METHOD PROTECTED M_MeasurementClient : BOOL
VAR_INPUT
END_VAR
CASE eFixtureStateMeasure OF
	UNIVERSAL_FIXTURE_MEASURE_SEND_DATA:
		(* Prepare and send data to client *)
		sSendData := CONCAT('START;',UDINT_TO_STRING(iSampleID));
		sSendData := CONCAT(sSendData, '$R$N');
		FUN_StringToTcpBufferData(sMessageAddr := ADR(sSendData), stSendDataAddr := ADR(stSendData));
		fbTcpClient.MR_AppendToSendBuffer(stData := stSendData);
		
		(* Prepare data for logger *)
		IF bUseLogger THEN
			MEMSET(ADR(sLoggerMessage),0,INT_TO_UDINT(LEN(sLoggerMessage)));
			sLoggerMessage := CONCAT('SampleID:',UDINT_TO_STRING(iSampleID));
			
		END_IF
		
		eFixtureStateMeasure := UNIVERSAL_FIXTURE_MEASURE_RECIVE_DATA;
		
	UNIVERSAL_FIXTURE_MEASURE_RECIVE_DATA:
		stReciveData := fbTcpClient.NextRecivedMessage;
		
		IF stReciveData.iLength > 0 THEN
			FUN_TcpBufferDataToString(sMessageAddr := ADR(sRecivedData), stReturnDataAddr := ADR(stReciveData));
			
			(* Sample accepted *)
			IF MEMCMP(ADR(sRecivedData),ADR(sSAMPLE_ACCEPTED),INT_TO_UDINT(LEN(sSAMPLE_ACCEPTED))) = 0 THEN
				IF bUseLogger THEN
					sLoggerMessage := CONCAT(sLoggerMessage,sSAMPLE_ACCEPTED);
					fbMeasurementLogger.MR_AddLogs(sLoggerMessage);
					
				END_IF
				eSampleResult := UNIVERSAL_FIXTURE_SAMPLE_ACCEPTED;
				eFixtureStateMeasure := UNIVERSAL_FIXTURE_MEASURE_DONE;
				
			(* Sample rejected *)
			ELSIF MEMCMP(ADR(sRecivedData),ADR(sSAMPLE_REJECTED),INT_TO_UDINT(LEN(sSAMPLE_REJECTED))) = 0 THEN
				IF bUseLogger THEN
					sLoggerMessage := CONCAT(sLoggerMessage,sSAMPLE_REJECTED);
					fbMeasurementLogger.MR_AddLogs(sLoggerMessage);
					
				END_IF
				eSampleResult := UNIVERSAL_FIXTURE_SAMPLE_REJECTED;
				eFixtureStateMeasure := UNIVERSAL_FIXTURE_MEASURE_DONE;
				
			END_IF
		END_IF
		
	UNIVERSAL_FIXTURE_MEASURE_DONE:
		fbTcpClient.MR_ClearAllBuffers();
		eFixtureStateMeasure := UNIVERSAL_FIXTURE_MEASURE_SEND_DATA;
		eFixtureState := UNIVERSAL_FIXTURE_METHOD_DONE;
		
END_CASE
END_METHOD

METHOD PROTECTED M_MeasurementServer : BOOL
VAR_INPUT
END_VAR
CASE eFixtureStateMeasure OF
	UNIVERSAL_FIXTURE_MEASURE_WAIT_FOR_CLIENT:
		IF fbTcpServer.ServerState = TCPIP_SERVER_RUNNING_DATA_EXCHANGE THEN
			eFixtureStateMeasure := UNIVERSAL_FIXTURE_MEASURE_SEND_DATA;
		END_IF
		
	UNIVERSAL_FIXTURE_MEASURE_SEND_DATA:
		(* Prepare and send data to client *)
		sSendData := CONCAT('START;',UDINT_TO_STRING(iSampleID));
		sSendData := CONCAT(sSendData, '$R$N');
		FUN_StringToTcpBufferData(sMessageAddr := ADR(sSendData), stSendDataAddr := ADR(stSendData));
		fbTcpServer.MR_AppendToSendBuffer(stData := stSendData);
		
		(* Prepare data for logger *)
		IF bUseLogger THEN
			MEMSET(ADR(sLoggerMessage),0,INT_TO_UDINT(LEN(sLoggerMessage)));
			sLoggerMessage := CONCAT('SampleID:',UDINT_TO_STRING(iSampleID));
		END_IF
		
		eFixtureStateMeasure := UNIVERSAL_FIXTURE_MEASURE_RECIVE_DATA;
		
	UNIVERSAL_FIXTURE_MEASURE_RECIVE_DATA:
		stReciveData := fbTcpServer.LastRecivedMessage;
		IF stReciveData.iLength > 0 THEN
			FUN_TcpBufferDataToString(sMessageAddr := ADR(sRecivedData), stReturnDataAddr := ADR(stReciveData));
			
			(* Sample accepted *)
			IF MEMCMP(ADR(sRecivedData),ADR(sSAMPLE_ACCEPTED),INT_TO_UDINT(LEN(sSAMPLE_ACCEPTED))) = 0 THEN
				IF bUseLogger THEN
					sLoggerMessage := CONCAT(sLoggerMessage,sSAMPLE_ACCEPTED);
					fbMeasurementLogger.MR_AddLogs(sLoggerMessage);
				END_IF
				eSampleResult := UNIVERSAL_FIXTURE_SAMPLE_ACCEPTED;
				eFixtureStateMeasure := UNIVERSAL_FIXTURE_MEASURE_DONE;
				
			(* Sample rejected *)
			ELSIF MEMCMP(ADR(sRecivedData),ADR(sSAMPLE_REJECTED),INT_TO_UDINT(LEN(sSAMPLE_REJECTED))) = 0 THEN
				IF bUseLogger THEN
					sLoggerMessage := CONCAT(sLoggerMessage,sSAMPLE_REJECTED);
					fbMeasurementLogger.MR_AddLogs(sLoggerMessage);
				END_IF
				eSampleResult := UNIVERSAL_FIXTURE_SAMPLE_REJECTED;
				eFixtureStateMeasure := UNIVERSAL_FIXTURE_MEASURE_DONE;
				
			END_IF
		END_IF
		
	UNIVERSAL_FIXTURE_MEASURE_DONE:
		fbTcpServer.MR_ClearAllBuffers();
		eFixtureStateMeasure := UNIVERSAL_FIXTURE_MEASURE_WAIT_FOR_CLIENT;
		eFixtureState := UNIVERSAL_FIXTURE_METHOD_DONE;
		
END_CASE
END_METHOD

METHOD MR_Abort : BOOL
IF eFixtureState >= UNIVERSAL_FIXTURE_INITIALIZING THEN
	bBusy := TRUE;
	MR_Abort := FALSE;
	eFixtureState := UNIVERSAL_FIXTURE_ABORTING;
	fbMachineLogger.MR_AddLogs(CONCAT(sName,' : abort requested'));	

ELSIF eFixtureState = UNIVERSAL_FIXTURE_UNINITIALIZED THEN
	bBusy := FALSE;
	MR_Abort := TRUE;
	fbMachineLogger.MR_AddLogs(CONCAT(sName,' : abort done'));	

END_IF
END_METHOD

METHOD MR_Close : BOOL
IF eFixtureState = UNIVERSAL_FIXTURE_IDLE AND THIS^.SocketOpen THEN
	bBusy := TRUE;	
	MR_Close := FALSE;
	eFixtureState := UNIVERSAL_FIXTURE_CLOSE;
	fbMachineLogger.MR_AddLogs(CONCAT(sName,' : close requested'));	
	
ELSIF eFixtureState = UNIVERSAL_FIXTURE_METHOD_DONE THEN
	bBusy := FALSE;
	MR_Close := TRUE;
	fbMachineLogger.MR_AddLogs(CONCAT(sName,' : close done'));	

END_IF
END_METHOD

METHOD MR_FirstCycle : BOOL
VAR_INPUT
	sFixtureName 		: STRING;		(*  *)
	sHost				: T_IPv4Addr;	(*  *)
	sAmsNetID 			: T_AmsNetID;	(*  *)
	iPort				: UINT;			(*  *)
	tTimeout			: TIME;			(*  *)
	bUseLogger			: BOOL;			(*  *)
	bClientConnection 	: BOOL;			(*  *)
	sFileDir			: STRING;		(*  *)
	sFileName			: STRING;		(*  *)
	bCreateFileAtStart	: BOOL;
	bAddHeader			: BOOL;
	bAddTimeStamp		: BOOL;	
END_VAR
THIS^.sName := sFixtureName;
THIS^.bUseLogger := bUseLogger;
THIS^.bClientConnection := bClientConnection;

IF THIS^.bClientConnection THEN 
	(* Set fixture client initial parameters *)
	THIS^.fbTcpClient.MR_FirstCycle(	sName 		:= CONCAT('TCP/IP client of ',sFixtureName),
										sHost		:= sHost,
										sAmsNetID	:= sAmsNetID,
										iPort 		:= iPort,
										tTimeout 	:= tTimeout);	
ELSE
	(* Set fixture server initial parameters *)
	THIS^.fbTcpServer.MR_FirstCycle(	sName 		:= CONCAT('TCP/IP server of ',sFixtureName),
										sHost		:= sHost,
										sAmsNetID	:= sAmsNetID,
										iPort 		:= iPort,
										tTimeout 	:= tTimeout);
END_IF								
									
IF THIS^.bUseLogger THEN
	(* Set measurement logger initial parameters*)									
	THIS^.fbMeasurementLogger.MR_FirstCycle(sName 	:= sName,
											sFileDir 	:= sFileDir,
											sFileName 	:= sFileName,
											sAmsNetId 	:= '',
											bCreateFileAtStart := bCreateFileAtStart,
											bAddHeader 	:= bAddHeader,
											bAddTimeStamp := bAddTimeStamp);	
END_IF
END_METHOD

METHOD MR_Init : BOOL
IF eFixtureState = UNIVERSAL_FIXTURE_UNINITIALIZED THEN
	bBusy := TRUE;
	MR_Init := FALSE;
	
	IF bClientConnection THEN 
		eConnnectionType := UNIVERSAL_FIXTURE_CLIENT_CONNECTION;
		eFixtureStateInit := UNIVERSAL_FIXTURE_INIT_TCP_CLIENT;
		
	ELSE
		eConnnectionType := UNIVERSAL_FIXTURE_SERVER_CONNECTION;	
		eFixtureStateInit := UNIVERSAL_FIXTURE_INIT_TCP_SERVER;	
		
	END_IF
	
	eFixtureState := UNIVERSAL_FIXTURE_INITIALIZING;
	fbMachineLogger.MR_AddLogs(CONCAT(sName,' : initialization requested'));	
	
ELSIF eFixtureState >= UNIVERSAL_FIXTURE_READY THEN
	bBusy := FALSE;
	MR_Init := TRUE;
	fbMachineLogger.MR_AddLogs(CONCAT(sName,' : initialization done'));
	
END_IF
END_METHOD

METHOD MR_Measure : BOOL
VAR_INPUT
	iSampleID : UINT;
END_VAR
IF eFixtureState = UNIVERSAL_FIXTURE_IDLE THEN
	bBusy := TRUE;
	MR_Measure := FALSE;
	THIS^.iSampleID := iSampleID;
	THIS^.eSampleResult := UNIVERSAL_FIXTURE_SAMPLE_UNKNOWN;
	
	IF eConnnectionType = UNIVERSAL_FIXTURE_SERVER_CONNECTION THEN
		eFixtureStateMeasure := UNIVERSAL_FIXTURE_MEASURE_WAIT_FOR_CLIENT;
		
	ELSIF eConnnectionType = UNIVERSAL_FIXTURE_CLIENT_CONNECTION THEN
		eFixtureStateMeasure := UNIVERSAL_FIXTURE_MEASURE_SEND_DATA;
		
	END_IF
	
	eFixtureState := UNIVERSAL_FIXTURE_MEASUREMENT;
	fbMachineLogger.MR_AddLogs(CONCAT(sName,' : measurement requested'));	

ELSIF eFixtureState = UNIVERSAL_FIXTURE_METHOD_DONE THEN
	bBusy := FALSE;
	MR_Measure := TRUE;
	fbMachineLogger.MR_AddLogs(CONCAT(sName,' : measurement done'));	
	
END_IF
END_METHOD

METHOD MR_Open : BOOL
IF eFixtureState = UNIVERSAL_FIXTURE_IDLE AND NOT THIS^.SocketOpen THEN
	bBusy := TRUE;
	MR_Open := FALSE;
	eFixtureState := UNIVERSAL_FIXTURE_OPEN;
	fbMachineLogger.MR_AddLogs(CONCAT(sName,' : open requested'));		
	
ELSIF eFixtureState = UNIVERSAL_FIXTURE_METHOD_DONE THEN
	bBusy := FALSE;
	MR_Open := TRUE;
	fbMachineLogger.MR_AddLogs(CONCAT(sName,' : open done'));		
	
END_IF
END_METHOD

METHOD MR_Reset : BOOL
IF eFixtureState >= UNIVERSAL_FIXTURE_IDLE AND bError THEN
	bBusy := TRUE;
	MR_Reset := FALSE;
	eFixtureState := UNIVERSAL_FIXTURE_RESET;
	fbMachineLogger.MR_AddLogs(CONCAT(sName,' : reset requested'));			
	
ELSIF eFixtureState = UNIVERSAL_FIXTURE_METHOD_DONE THEN
	bBusy := FALSE;
	MR_Reset := TRUE;
	fbMachineLogger.MR_AddLogs(CONCAT(sName,' : reset done'));			
	
END_IF
END_METHOD

METHOD PROTECTED MS_Aborting
VAR_INPUT
END_VAR
CASE eFixtureStateAbort OF
	UNIVERSAL_FIXTURE_ABORT_FILE_LOGGER:
		IF bUseLogger THEN
			fbMeasurementLogger.MR_Abort();
		
			IF NOT fbMeasurementLogger.Busy THEN
				IF eConnnectionType = UNIVERSAL_FIXTURE_SERVER_CONNECTION THEN
					eFixtureStateAbort := UNIVERSAL_FIXTURE_ABORT_TCP_SERVER;
					
				ELSIF eConnnectionType = UNIVERSAL_FIXTURE_CLIENT_CONNECTION THEN
					eFixtureStateAbort := UNIVERSAL_FIXTURE_ABORT_TCP_CLIENT;
					
				END_IF
			END_IF
		ELSE
			IF eConnnectionType = UNIVERSAL_FIXTURE_SERVER_CONNECTION THEN
				eFixtureStateAbort := UNIVERSAL_FIXTURE_ABORT_TCP_SERVER;
				
			ELSIF eConnnectionType = UNIVERSAL_FIXTURE_CLIENT_CONNECTION THEN
				eFixtureStateAbort := UNIVERSAL_FIXTURE_ABORT_TCP_CLIENT;
				
			END_IF
		END_IF
		
	UNIVERSAL_FIXTURE_ABORT_TCP_SERVER:
		fbTcpServer.MR_Abort();
		
		IF NOT fbTcpServer.Active THEN
			eFixtureStateAbort := UNIVERSAL_FIXTURE_ABORT_DONE;
			
		END_IF

	UNIVERSAL_FIXTURE_ABORT_TCP_CLIENT:
		fbTcpClient.MR_Abort();
		
		IF NOT fbTcpClient.Active THEN
			eFixtureStateAbort := UNIVERSAL_FIXTURE_ABORT_DONE;
			
		END_IF
		
	UNIVERSAL_FIXTURE_ABORT_DONE:
		eFixtureStateAbort := UNIVERSAL_FIXTURE_ABORT_FILE_LOGGER;
		eFixtureState := UNIVERSAL_FIXTURE_UNINITIALIZED;
	
END_CASE
END_METHOD

METHOD PROTECTED ABSTRACT MS_Close
VAR_INPUT
END_VAR
;
END_METHOD

METHOD PROTECTED MS_Extension
VAR_INPUT
END_VAR
END_METHOD

METHOD PROTECTED MS_Idle
VAR_INPUT
END_VAR
;
END_METHOD

METHOD PROTECTED MS_Initializing
VAR_INPUT
END_VAR
CASE eFixtureStateInit OF
	UNIVERSAL_FIXTURE_INIT_TCP_SERVER:
		fbTcpServer.MR_Init();
		
		IF fbTcpServer.Active THEN
			eFixtureStateInit := UNIVERSAL_FIXTURE_INIT_FILE_LOGGER;
			
		END_IF

	UNIVERSAL_FIXTURE_INIT_TCP_CLIENT:
		fbTcpClient.MR_Init();
		
		IF fbTcpClient.Active THEN
			eFixtureStateInit := UNIVERSAL_FIXTURE_INIT_FILE_LOGGER;
			
		END_IF
		
	UNIVERSAL_FIXTURE_INIT_FILE_LOGGER:
		IF bUseLogger THEN
			fbMeasurementLogger.MR_Init();
		
			IF fbMeasurementLogger.Busy THEN
				eFixtureStateInit := UNIVERSAL_FIXTURE_INIT_DONE;
				
			END_IF
		ELSE
			eFixtureStateInit := UNIVERSAL_FIXTURE_INIT_DONE;
			
		END_IF
		
	UNIVERSAL_FIXTURE_INIT_DONE:
		eFixtureStateInit := UNIVERSAL_FIXTURE_INIT_TCP_SERVER;
		eFixtureState := UNIVERSAL_FIXTURE_READY;
	
END_CASE
END_METHOD

METHOD PROTECTED MS_Measurement
VAR_INPUT
END_VAR
IF eConnnectionType = UNIVERSAL_FIXTURE_SERVER_CONNECTION THEN
	M_MeasurementServer();
	
ELSIF eConnnectionType = UNIVERSAL_FIXTURE_CLIENT_CONNECTION THEN
	M_MeasurementClient();
	
END_IF
END_METHOD

METHOD PROTECTED MS_MethodDone
VAR_INPUT
END_VAR
IF NOT bBusy THEN
	eFixtureState := UNIVERSAL_FIXTURE_IDLE;
	
END_IF
END_METHOD

METHOD PROTECTED ABSTRACT MS_Open
VAR_INPUT
END_VAR
END_METHOD

METHOD PROTECTED MS_Ready
VAR_INPUT
END_VAR
eFixtureState := UNIVERSAL_FIXTURE_IDLE;
END_METHOD

METHOD PROTECTED MS_Reset
VAR_INPUT
END_VAR
CASE eFixtureStateReset OF 
	UNIVERSAL_FIXTURE_RESETING_FILE_LOGGER:
		IF bUseLogger THEN
			fbMeasurementLogger.MR_Reset();
		
			IF NOT fbMeasurementLogger.Busy THEN
				IF eConnnectionType = UNIVERSAL_FIXTURE_SERVER_CONNECTION THEN
					eFixtureStateReset := UNIVERSAL_FIXTURE_RESETING_TCP_SERVER_SHUT_DOWN;
					
				ELSIF eConnnectionType = UNIVERSAL_FIXTURE_CLIENT_CONNECTION THEN
					eFixtureStateReset := UNIVERSAL_FIXTURE_RESETING_TCP_CLIENT_SHUT_DOWN;
					
				END_IF
			END_IF
		ELSE
			IF eConnnectionType = UNIVERSAL_FIXTURE_SERVER_CONNECTION THEN
				eFixtureStateReset := UNIVERSAL_FIXTURE_RESETING_TCP_SERVER_SHUT_DOWN;
				
			ELSIF eConnnectionType = UNIVERSAL_FIXTURE_CLIENT_CONNECTION THEN
				eFixtureStateReset := UNIVERSAL_FIXTURE_RESETING_TCP_CLIENT_SHUT_DOWN;
				
			END_IF
		END_IF
		
	UNIVERSAL_FIXTURE_RESETING_TCP_SERVER_SHUT_DOWN:
		fbTcpServer.MR_Abort();
		
		IF NOT fbTcpServer.Active THEN
			eFixtureStateReset := UNIVERSAL_FIXTURE_RESETING_TCP_SERVER_TURN_ON;
			
		END_IF
		
	UNIVERSAL_FIXTURE_RESETING_TCP_SERVER_TURN_ON:
		fbTcpServer.MR_Init();
		
		IF fbTcpServer.Active THEN
			eFixtureStateReset := UNIVERSAL_FIXTURE_RESETING_DONE;
			
		END_IF

	UNIVERSAL_FIXTURE_RESETING_TCP_CLIENT_SHUT_DOWN:
		fbTcpClient.MR_Abort();
		
		IF NOT fbTcpClient.Active THEN
			eFixtureStateReset := UNIVERSAL_FIXTURE_RESETING_TCP_CLIENT_TURN_ON;
			
		END_IF
		
	UNIVERSAL_FIXTURE_RESETING_TCP_CLIENT_TURN_ON:
		fbTcpClient.MR_Init();
		
		IF fbTcpClient.Active THEN
			eFixtureStateReset := UNIVERSAL_FIXTURE_RESETING_DONE;
			
		END_IF
		
	UNIVERSAL_FIXTURE_RESETING_DONE:		
		bError := FALSE;
		
		eFixtureStateReset := UNIVERSAL_FIXTURE_RESETING_FILE_LOGGER;
		eFixtureState := UNIVERSAL_FIXTURE_METHOD_DONE;
		
END_CASE
END_METHOD

METHOD PROTECTED MS_Uninitialized
VAR_INPUT
END_VAR
bBusy := FALSE;
bError := FALSE;
iErrorID := 0;
iSampleID := 0;

eSampleResult := UNIVERSAL_FIXTURE_SAMPLE_UNKNOWN;
END_METHOD

PROPERTY RecivedUtuData : REFERENCE TO STRING
GET
RecivedUtuData REF= sRecivedData;
END_GET
END_PROPERTY

PROPERTY ref_MeasurementLogger : REFERENCE TO FB_TXTDataExchanger
GET
ref_MeasurementLogger REF= fbMeasurementLogger;
END_GET
END_PROPERTY

PROPERTY ref_TcpClient : REFERENCE TO FB_TcpClient
GET
ref_TcpClient REF= fbTcpClient;
END_GET
END_PROPERTY

PROPERTY ref_TcpServer : REFERENCE TO FB_TcpServer
GET
ref_TcpServer REF= fbTcpServer;
END_GET
END_PROPERTY

PROPERTY SampleID : REFERENCE TO UDINT
GET
SampleID REF= iSampleID;
END_GET
END_PROPERTY

PROPERTY SampleResult : REFERENCE TO E_UniversalFixtureSampleResult
GET
SampleResult REF= eSampleResult;
END_GET
END_PROPERTY

PROPERTY ABSTRACT SocketOpen : REFERENCE TO BOOL
GET
END_GET
END_PROPERTY

PROPERTY State : REFERENCE TO E_UniversalFixtureState
GET
State REF= eFixtureState;
END_GET
END_PROPERTY

METHOD PROTECTED StateMachine
VAR_INPUT
END_VAR
CASE eFixtureState OF
	UNIVERSAL_FIXTURE_UNINITIALIZED:
		MS_Uninitialized();
		
	UNIVERSAL_FIXTURE_INITIALIZING:
		MS_Initializing();
		
	UNIVERSAL_FIXTURE_READY:
		MS_Ready();
		
	UNIVERSAL_FIXTURE_IDLE:
		MS_Idle();
	
	UNIVERSAL_FIXTURE_OPEN:
		MS_Open();
		
	UNIVERSAL_FIXTURE_CLOSE:
		MS_Close();
	
	UNIVERSAL_FIXTURE_MEASUREMENT:
		MS_Measurement();
	
	UNIVERSAL_FIXTURE_RESET:
		MS_Reset();
		
	UNIVERSAL_FIXTURE_METHOD_DONE:
		MS_MethodDone();
		
	UNIVERSAL_FIXTURE_EXTENSION:
		MS_Extension();
	
	UNIVERSAL_FIXTURE_ABORTING:
		MS_Aborting();
	
END_CASE
END_METHOD

END_FUNCTION_BLOCK

// ---- POUs/Libs/Utilities/TXT Data Exchanger/FB_TXTDataExchanger.TcPOU
FUNCTION_BLOCK FB_TXTDataExchanger IMPLEMENTS I_TXTDataExchanger
VAR CONSTANT
	iBUFFER_SIZE 						: UINT := 255;
END_VAR
VAR
	sName : STRING;
	
	(* First cycle bits used for selecting file logging mode *)
	bAddTimeStamp						: BOOL;
	bAddHeader							: BOOL;
	bCreateFileAtStart					: BOOL;    
                        		
	(* Internal status *)       		
	bActive 							: BOOL;										(*  *)
	bBusy								: BOOL;										(*  *)
	bError								: BOOL;										(*  *)
	iErrorID							: UDINT;									(*  *)
	                                                                            	
	eTXTDataExchangerState 				: E_TXTDataExchangerState;					(*  *)
	eTXTDataExchangerInitState 			: E_TXTDataExchangerInitState;				(*  *)
	eTXTDataExchangerAddLogsState		: E_TXTDataExchangerAddLogsState; 			(*  *)
	eTXTDataExchangerSetNewPathState 	: E_TXTDataExchangerSetNewPathState;
	eTXTDataExchangerSearchForFileState : E_TXTDataExchangerSearchForFileState;
	
	(* Internal parameters *)
	sFileName 							: STRING;									(*  *)
	sFileDir							: STRING;									(*  *)
	sFilePath							: STRING;									(*  *)
                   				      		
	hFile								: UINT;										(*  *)

	sAmsNetId							: T_AmsNetID;								(*  *)
	stTime								: TIMESTRUCT;								(*  *)
	sTime								: STRING;									(*  *)
	sFileDate							: STRING;									(*  *)

	sLogMessage							: STRING;									(*  *)

	sSearchFileName						: STRING; 
	bFileFound							: BOOL;                       		
	
	(* Buffer arrays *)         		
	iCurrentBufferLine					: UINT := 1;								(*  *)
	iCurrentBufferLineForFile			: UINT := 1;								(*  *)
	arrMessageBuffer 					: ARRAY [1..iBUFFER_SIZE] OF STRING(300);	(*  *)
	arrMessageBufferPresence			: ARRAY [1..iBUFFER_SIZE] OF BOOL(255);		(*  *)
	
	(* Function blocks - file handling *)
	fbFileOpen							: FB_FileOpen;								(*  *)
	fbFileClose							: FB_FileClose;								(*  *)
	fbCreateDir							: FB_CreateDir;								(*  *)
	fbFilePuts							: FB_FilePuts;								(*  *)
	fbEnumFindFileEntry					: FB_EnumFindFileEntry;
END_VAR

bActive := eTXTDataExchangerState >= TXT_DATA_EXCHANGER_READY;

IF fbMachineTime.bValid THEN
	stTime := fbMachineTime.systemTime;
	sTime := SYSTEMTIME_TO_STRING(stTime);
	
END_IF

StateMachine();

PROPERTY Active : REFERENCE TO BOOL
GET
Active REF= bActive;
END_GET
END_PROPERTY

PROPERTY AmsNetId : STRING
GET
AmsNetID := sAmsNetId;
END_GET
SET
sAmsNetId := AmsNetId;
END_SET
END_PROPERTY

PROPERTY Busy : REFERENCE TO BOOL
GET
Busy REF= bBusy;
END_GET
END_PROPERTY

PROPERTY Error : REFERENCE TO BOOL
GET
Error REF= bError;
END_GET
END_PROPERTY

PROPERTY ErrorID : REFERENCE TO UDINT
GET
ErrorID REF= iErrorID;
END_GET
END_PROPERTY

PROPERTY FileDir : STRING
GET
FileDir := sFileDir;
END_GET
SET
sFileDir := FileDir;
END_SET
END_PROPERTY

PROPERTY FileName : STRING
GET
FileName := sFileName;
END_GET
SET
sFileName := FileName;
END_SET
END_PROPERTY

METHOD M_ResetParameters : BOOL
VAR_INPUT
END_VAR
fbCreateDir( bExecute := FALSE);
fbFileOpen( bExecute := FALSE);
fbFilePuts( bExecute := FALSE);
fbFileClose( bExecute := FALSE);

FOR iCurrentBufferLine := 1 TO iBUFFER_SIZE BY 1 DO
	MEMSET(ADR(arrMessageBuffer[iCurrentBufferLine]),0,SIZEOF(arrMessageBuffer[iCurrentBufferLine]));
	arrMessageBufferPresence[iCurrentBufferLine] := FALSE;
END_FOR

iCurrentBufferLine := 1;
iCurrentBufferLineForFile := 1;

bError 		:= FALSE;
iErrorID 	:= 0;

MEMSET(ADR(sLogMessage),0,SIZEOF(sLogMessage));

eTXTDataExchangerInitState := 0;
eTXTDataExchangerAddLogsState := 0;
END_METHOD

METHOD M_SetNewPath : BOOL
VAR_INPUT
END_VAR
CASE eTXTDataExchangerSetNewPathState OF
	TXT_DATA_EXCHANGER_SET_NEW_PATH_CHANGE_PATH:
		M_SetNewPath := FALSE;
		sFilePath := FUN_MergeStrings3(sStr1 := sFileDir, sStr2 := sFileName, sStr3 :=  '.txt');
		eTXTDataExchangerSetNewPathState := TXT_DATA_EXCHANGER_SET_NEW_PATH_DONE;
	
	TXT_DATA_EXCHANGER_SET_NEW_PATH_DONE:
		M_SetNewPath := TRUE;
		eTXTDataExchangerSetNewPathState := TXT_DATA_EXCHANGER_SET_NEW_PATH_CHANGE_PATH;
			
END_CASE
END_METHOD

METHOD MR_Abort : BOOL
IF eTXTDataExchangerState >= TXT_DATA_EXCHANGER_READY THEN
	bBusy := TRUE;
	MR_Abort := FALSE;
	eTXTDataExchangerState := TXT_DATA_EXCHANGER_ABORTING;
	
ELSIF eTXTDataExchangerState = TXT_DATA_EXCHANGER_UNINITIALIZED THEN
	bBusy := FALSE;
	MR_Abort := TRUE;
	
END_IF
END_METHOD

METHOD MR_AddLogs : BOOL
VAR_INPUT
	sLogMessage 	: STRING;		
	
END_VAR
VAR
	sCurrentTime 	: STRING;
	sCurrentDate	: STRING;
	sLog			: STRING(300);
	
END_VAR
IF iCurrentBufferLine >= iBUFFER_SIZE THEN	
	iCurrentBufferLine := 1;
		
ELSE
	sCurrentDate := LEFT(sTime,10);
	sCurrentTime := RIGHT(sTime,12);
	MEMSET(ADR(sLog),0,SIZEOF(sLog));
	
	IF bAddTimeStamp THEN
		sLog := FUN_MergeStrings6(sCurrentDate,'$t',sCurrentTime,'$t',sLogMessage,'$n'); 
	ELSE
		sLog := CONCAT(sLogMessage,'$n'); 
	END_IF
	
	MEMSET(ADR(arrMessageBuffer[iCurrentBufferLine]),0,SIZEOF(arrMessageBuffer[iCurrentBufferLine]));
	arrMessageBuffer[iCurrentBufferLine] := sLog;
	iCurrentBufferLine := iCurrentBufferLine + 1;
	
	MR_AddLogs := TRUE;
	
END_IF
END_METHOD

METHOD MR_AddMESCommand : BOOL
VAR_INPUT
	sMachineID		: STRING;
	sOperatorID		: STRING;
	sPO				: STRING;
	sProductItem	: STRING;
	bLogOn			: BOOL;
END_VAR

VAR
	sLog			: STRING(300);
END_VAR
IF iCurrentBufferLine >= iBUFFER_SIZE THEN	
	iCurrentBufferLine := 1;
		
ELSE
	MEMSET(ADR(sLog),0,SIZEOF(sLog));

	IF bLogOn THEN
		sLog := FUN_MergeStrings10(sStr1 := 'DLG=A_P_AN|MNR=', 
									sStr2 := sMachineID,
									sStr3 := '|KNR=',
									sStr4 := sOperatorID,
									sStr5 := '|AUNR=',
									sStr6 := sPO,									
									sStr7 := '|ATK=',
									sStr8 := sProductItem,
									sStr9 := '|M_HS=1',
									sStr10 :='$n');  
									
	ELSE
		sLog := FUN_MergeStrings10(sStr1 := 'DLG=A_AB|MNR=', 
									sStr2 := sMachineID,
									sStr3 := '|KNR=',
									sStr4 := sOperatorID,
									sStr5 := '|AUNR=',
									sStr6 := sPO,									
									sStr7 := '|ATK=',
									sStr8 := sProductItem,
									sStr9 := '|M_HS=2',
									sStr10 :='$n');  
									
	END_IF
	
	MEMSET(ADR(arrMessageBuffer[iCurrentBufferLine]),0,SIZEOF(arrMessageBuffer[iCurrentBufferLine]));
	arrMessageBuffer[iCurrentBufferLine] := sLog;
	iCurrentBufferLine := iCurrentBufferLine + 1;
	
	MR_AddMESCommand := TRUE;
	
END_IF
END_METHOD

METHOD MR_FirstCycle : BOOL
VAR_INPUT
	sName 					: STRING;
	sFileDir				: STRING(255);
	sFileName				: STRING(255);
	sAmsNetId				: T_AmsNetID;		
	bAddTimeStamp			: BOOL;				(* If true the time stamp will be added to each log *)
	bAddHeader				: BOOL;				(* If true the header will be added to the file at the start-up *)
	bCreateFileAtStart		: BOOL;				(* If true the file will be created at the start-up *)
END_VAR
THIS^.sName := sName;
THIS^.sFileDir := sFileDir;
THIS^.sFileName := sFileName;
THIS^.sAmsNetId := sAmsNetId;
THIS^.bAddTimeStamp := bAddTimeStamp;
THIS^.bAddHeader := bAddHeader;
THIS^.bCreateFileAtStart := bCreateFileAtStart;

M_SetNewPath();
END_METHOD

METHOD MR_Init : BOOL
VAR_INPUT
END_VAR
IF eTXTDataExchangerState = TXT_DATA_EXCHANGER_UNINITIALIZED THEN
	bBusy := TRUE;
	MR_Init := FALSE;
	eTXTDataExchangerState := TXT_DATA_EXCHANGER_INITIALIZING;
	
ELSIF eTXTDataExchangerState >= TXT_DATA_EXCHANGER_READY THEN
	bBusy := FALSE;
	MR_Init := TRUE;
	
END_IF
END_METHOD

METHOD MR_Reset : BOOL
IF eTXTDataExchangerState >= TXT_DATA_EXCHANGER_IDLE AND eTXTDataExchangerState <> TXT_DATA_EXCHANGER_METHOD_DONE THEN
	bBusy := TRUE;
	MR_Reset := FALSE;
	eTXTDataExchangerState := TXT_DATA_EXCHANGER_RESET;	

ELSIF eTXTDataExchangerState = TXT_DATA_EXCHANGER_METHOD_DONE THEN
	bBusy := FALSE;
	MR_Reset := TRUE;

END_IF
END_METHOD

METHOD MR_SearchForFile : BOOL
VAR_INPUT
	sSearchFileName		: STRING;			(* Whole name of the search file (e.g.: "DemoFile.txt" *)
END_VAR

VAR_OUTPUT
	bFileFound	: BOOL;
END_VAR
IF eTXTDataExchangerState = TXT_DATA_EXCHANGER_IDLE THEN
	THIS^.sSearchFileName := sSearchFileName;
	bFileFound	:= FALSE;
	bBusy := TRUE;
	MR_SearchForFile := FALSE;
	eTXTDataExchangerState := TXT_DATA_EXCHANGER_SEARCH_FOR_FILE;
	
ELSIF eTXTDataExchangerState = TXT_DATA_EXCHANGER_METHOD_DONE THEN
	bFileFound := THIS^.bFileFound;
	bBusy := FALSE;
	MR_SearchForFile := TRUE;
	
END_IF
END_METHOD

METHOD MR_SelectPath : BOOL
VAR_INPUT
	sFileDir								: STRING; 			(* CSV source file directory name *)
	sFileName 								: STRING; 			(* CSV source file name *)
END_VAR
IF eTXTDataExchangerState = TXT_DATA_EXCHANGER_IDLE THEN
	THIS^.sFileDir := sFileDir;	
	THIS^.sFileName := sFileName;	
	bBusy := TRUE;
	MR_SelectPath := FALSE;
	eTXTDataExchangerState := TXT_DATA_EXCHANGER_SELECT_PATH;
	
ELSIF eTXTDataExchangerState = TXT_DATA_EXCHANGER_METHOD_DONE THEN
	bBusy := FALSE;
	MR_SelectPath := TRUE;
	
END_IF
END_METHOD

METHOD PROTECTED MS_Aborting
fbCreateDir( bExecute := FALSE);
fbFileOpen( bExecute := FALSE);
fbFilePuts( bExecute := FALSE);
fbFileClose( bExecute := FALSE);

FOR iCurrentBufferLine := 1 TO iBUFFER_SIZE BY 1 DO
	MEMSET(ADR(arrMessageBuffer[iCurrentBufferLine]),0,SIZEOF(arrMessageBuffer[iCurrentBufferLine]));
	arrMessageBufferPresence[iCurrentBufferLine] := FALSE;
	
END_FOR

iCurrentBufferLine := 1;
iCurrentBufferLineForFile := 1;

MEMSET(ADR(sTime),0,SIZEOF(sTime));
MEMSET(ADR(sFileDate),0,SIZEOF(sFileDate));
MEMSET(ADR(sLogMessage),0,SIZEOF(sLogMessage));

stTime.wDay 			:= 0;
stTime.wDayOfWeek 		:= 0;
stTime.wHour 			:= 0;
stTime.wMilliseconds 	:= 0;
stTime.wMinute 			:= 0;
stTime.wMonth 			:= 0;
stTime.wSecond 			:= 0;
stTime.wYear 			:= 0;

bActive		:= FALSE;
bBusy 		:= FALSE;
bError 		:= FALSE;
iErrorID 	:= 0;

eTXTDataExchangerInitState := TXT_DATA_EXCHANGER_INIT_GET_TIME;
eTXTDataExchangerAddLogsState := TXT_DATA_EXCHANGER_ADD_LOGS_OPEN;
eTXTDataExchangerState := TXT_DATA_EXCHANGER_UNINITIALIZED;
END_METHOD

METHOD PROTECTED MS_AddLogs
CASE eTXTDataExchangerAddLogsState OF
	TXT_DATA_EXCHANGER_ADD_LOGS_OPEN:
		IF NOT fbFileOpen.bError THEN
			fbFileOpen( sNetId 		:= sAmsNetId,
						sPathName 	:= sFilePath,
						bExecute 	:= TRUE,
						tTimeout	:= DEFAULT_ADS_TIMEOUT,
						nMode		:= FOPEN_MODEAPPEND OR FOPEN_MODEPLUS);
							
			IF NOT fbFileOpen.bBusy THEN
				fbFileOpen(bExecute := FALSE);				
				hFile := fbFileOpen.hFile;;
				eTXTDataExchangerAddLogsState := TXT_DATA_EXCHANGER_ADD_LOGS_WRITE;
			
			END_IF
		ELSE
			fbFileOpen( bExecute := FALSE);
			bError := fbFileOpen.bError;
			iErrorID := fbFileOpen.nErrId;

		END_IF
	

	TXT_DATA_EXCHANGER_ADD_LOGS_WRITE:
		IF NOT fbFilePuts.bError THEN
			fbFilePuts( sNetId		:= sAmsNetId,
						hFile 		:= hFile,
						sLine 		:= arrMessageBuffer[iCurrentBufferLineForFile],
						bExecute 	:= TRUE,
						tTimeout 	:= DEFAULT_ADS_TIMEOUT);	
					
			IF NOT fbFilePuts.bBusy THEN				
				eTXTDataExchangerAddLogsState := TXT_DATA_EXCHANGER_ADD_LOGS_WRITE_DONE;
				
			END_IF
			
		ELSE
			fbFilePuts( bExecute := FALSE);
			bError := fbFilePuts.bError;
			iErrorID := fbFilePuts.nErrId;
			
		END_IF	

		
	TXT_DATA_EXCHANGER_ADD_LOGS_WRITE_DONE:
		fbFilePuts( bExecute := FALSE);	
		iCurrentBufferLineForFile := iCurrentBufferLineForFile + 1;	
		
		IF iCurrentBufferLineForFile >= iBUFFER_SIZE THEN
			iCurrentBufferLineForFile := 1;
			
		ELSIF iCurrentBufferLineForFile < iCurrentBufferLine THEN
			eTXTDataExchangerAddLogsState := TXT_DATA_EXCHANGER_ADD_LOGS_WRITE;			
	
		ELSIF iCurrentBufferLineForFile >= iCurrentBufferLine THEN
			eTXTDataExchangerAddLogsState := TXT_DATA_EXCHANGER_ADD_LOGS_CLOSE;
			
		END_IF;

	
	TXT_DATA_EXCHANGER_ADD_LOGS_CLOSE:
		IF NOT fbFileClose.bError THEN
			fbFileClose(	sNetId := sAmsNetId,
							hFile := hFile,
							bExecute := TRUE,
							tTimeout := DEFAULT_ADS_TIMEOUT);
							
			IF NOT fbFileClose.bBusy THEN
				fbFileClose(bExecute := FALSE);
				eTXTDataExchangerAddLogsState := TXT_DATA_EXCHANGER_ADD_LOGS_OPEN;
				eTXTDataExchangerState := TXT_DATA_EXCHANGER_IDLE;

			END_IF
		ELSE
			bError := fbFileClose.bError;
			iErrorID := fbFileClose.nErrId;
			fbFileClose( bExecute := FALSE);
			
		END_IF
		
END_CASE
END_METHOD

METHOD PROTECTED MS_Idle
VAR_INPUT
END_VAR
IF iCurrentBufferLineForFile < iCurrentBufferLine THEN
	eTXTDataExchangerState := TXT_DATA_EXCHANGER_ADD_LOGS;

END_IF
END_METHOD

METHOD PROTECTED MS_Initializing //C:\TwinCAT\log\filelog.txt
CASE eTXTDataExchangerInitState OF
	TXT_DATA_EXCHANGER_INIT_CREATE_DIR:
		IF bCreateFileAtStart THEN
			fbCreateDir(sNetId 		:= sAmsNetId,
						sPathName 	:= sFileDir,
						bExecute 	:= TRUE,
						tTimeout 	:= DEFAULT_ADS_TIMEOUT);
						
			IF NOT fbCreateDir.bBusy THEN
				eTXTDataExchangerInitState := TXT_DATA_EXCHANGER_INIT_GET_TIME;
				fbCreateDir( bExecute := FALSE);
				
			END_IF
		ELSE
			eTXTDataExchangerInitState := TXT_DATA_EXCHANGER_INIT_DONE;
			
		END_IF
		
	TXT_DATA_EXCHANGER_INIT_GET_TIME:
		IF fbMachineTime.bValid THEN
			stTime := fbMachineTime.systemTime;
			sTime := SYSTEMTIME_TO_STRING(stTime);
			sFileDate := LEFT(sTime,10);
			eTXTDataExchangerInitState := TXT_DATA_EXCHANGER_INIT_CREATE_FILE;
			
		END_IF
		
	TXT_DATA_EXCHANGER_INIT_CREATE_FILE:
		IF NOT fbFileOpen.bError THEN
			fbFileOpen( sNetId 		:= sAmsNetId,
						sPathName 	:= sFilePath,
						bExecute 	:= TRUE,
						tTimeout	:= DEFAULT_ADS_TIMEOUT,
						nMode		:= FOPEN_MODEAPPEND OR FOPEN_MODEPLUS);
							
			IF NOT fbFileOpen.bBusy THEN
				hFile := fbFileOpen.hFile;
				fbFileOpen(bExecute := FALSE);		
				
				IF bAddHeader THEN 
					eTXTDataExchangerInitState := TXT_DATA_EXCHANGER_INIT_ADD_HEADER;
					
				ELSE
					eTXTDataExchangerInitState := TXT_DATA_EXCHANGER_INIT_CLOSE_FILE;
					
				END_IF							
			END_IF
		ELSE
			bError := fbFileOpen.bError;
			iErrorID := fbFileOpen.nErrId;
			fbFileOpen( bExecute := FALSE);
			
		END_IF
		
	TXT_DATA_EXCHANGER_INIT_ADD_HEADER:
		IF NOT fbFilePuts.bError THEN
			fbFilePuts(	sNetId := sAmsNetId,
						hFile := hFile,
						sLine := CONCAT('----- Logger file initialized at ',CONCAT(LEFT(sTime,23),' ----- $n')),
						bExecute := TRUE,
						tTimeout := DEFAULT_ADS_TIMEOUT);

			IF NOT fbFilePuts.bBusy THEN
				eTXTDataExchangerInitState := TXT_DATA_EXCHANGER_INIT_CLOSE_FILE;
				fbFilePuts( bExecute := FALSE);
				
			END_IF	
		ELSE
			bError := fbFilePuts.bError;
			iErrorID := fbFilePuts.nErrId;
			fbFilePuts( bExecute := FALSE);
			
		END_IF
	
	TXT_DATA_EXCHANGER_INIT_CLOSE_FILE:
		IF NOT fbFileClose.bError THEN
			fbFileClose( sNetId 		:= sAmsNetId,
							hFile 		:= hFile,
							bExecute 	:= TRUE,
							tTimeout 	:= DEFAULT_ADS_TIMEOUT);
							
			IF NOT fbFileClose.bBusy THEN
				eTXTDataExchangerInitState := TXT_DATA_EXCHANGER_INIT_DONE;
				fbFileClose( bExecute := FALSE);
				
			END_IF
		ELSE
			bError := fbFileClose.bError;
			iErrorID := fbFileClose.nErrId;
			fbFileClose( bExecute := FALSE);
			
		END_IF
	
	TXT_DATA_EXCHANGER_INIT_DONE:
		eTXTDataExchangerInitState := TXT_DATA_EXCHANGER_INIT_CREATE_DIR;
		eTXTDataExchangerState := TXT_DATA_EXCHANGER_IDLE;
		
END_CASE
END_METHOD

METHOD PROTECTED MS_MethodDone
VAR_INPUT
END_VAR
IF NOT bBusy THEN
	eTXTDataExchangerState := TXT_DATA_EXCHANGER_IDLE;

END_IF
END_METHOD

METHOD PROTECTED MS_Ready
VAR_INPUT
END_VAR
eTXTDataExchangerState := TXT_DATA_EXCHANGER_IDLE;
END_METHOD

METHOD PROTECTED MS_Reset
VAR_INPUT
END_VAR
IF M_ResetParameters() THEN
	eTXTDataExchangerState := TXT_DATA_EXCHANGER_METHOD_DONE;
	
END_IF
END_METHOD

METHOD MS_SearchForFile : BOOL
VAR_INPUT
END_VAR
CASE eTXTDataExchangerSearchForFileState OF
    TXT_DATA_EXCHANGER_SEARCH_FOR_FILE_ENUM_FIRST_ENTRY:
		bFileFound := FALSE;
		fbEnumFindFileEntry (sNetID := sAmsNetId, 
							 tTimeout := T#5S, 
							 sPathName := CONCAT(STR1 := sFileDir, STR2 := '*.*'));
		
		fbEnumFindFileEntry.eCmd := eEnumCmd_First;    (* enum first entry *)
		
		eTXTDataExchangerSearchForFileState := TXT_DATA_EXCHANGER_SEARCH_FOR_FILE_ENUM_NEXT_ENTRY;

    TXT_DATA_EXCHANGER_SEARCH_FOR_FILE_ENUM_NEXT_ENTRY:    (* enum one entry *)
        fbEnumFindFileEntry( bExecute := FALSE );
        fbEnumFindFileEntry( bExecute := TRUE );
		
        eTXTDataExchangerSearchForFileState := TXT_DATA_EXCHANGER_SEARCH_FOR_FILE_WAIT_FOR_READING;

    TXT_DATA_EXCHANGER_SEARCH_FOR_FILE_WAIT_FOR_READING:    (* wait until function block not busy *)
        fbEnumFindFileEntry( bExecute := FALSE );
		
        IF NOT fbEnumFindFileEntry.bBusy THEN
            IF NOT fbEnumFindFileEntry.bError THEN
                IF NOT fbEnumFindFileEntry.bEOE THEN
                   	IF sSearchFileName = fbEnumFindFileEntry.stFindFile.sFileName THEN
						bFileFound := TRUE;
						eTXTDataExchangerSearchForFileState := TXT_DATA_EXCHANGER_SEARCH_FOR_FILE_DONE;
						
					END_IF
                    fbEnumFindFileEntry.eCmd := eEnumCmd_Next; (* enum next entry *)
					
                    eTXTDataExchangerSearchForFileState := TXT_DATA_EXCHANGER_SEARCH_FOR_FILE_ENUM_NEXT_ENTRY;
					
                ELSE (* no more entries *)
                    eTXTDataExchangerSearchForFileState := TXT_DATA_EXCHANGER_SEARCH_FOR_FILE_DONE;
					
                END_IF
            ELSE (* log error *)       
				bError := fbEnumFindFileEntry.bError;
				iErrorID := fbEnumFindFileEntry.nErrID;
				eTXTDataExchangerSearchForFileState := TXT_DATA_EXCHANGER_SEARCH_FOR_FILE_DONE;
				
            END_IF
        END_IF
		
	TXT_DATA_EXCHANGER_SEARCH_FOR_FILE_DONE:
			eTXTDataExchangerSearchForFileState := TXT_DATA_EXCHANGER_SEARCH_FOR_FILE_ENUM_FIRST_ENTRY;
			eTXTDataExchangerState := TXT_DATA_EXCHANGER_METHOD_DONE;
		
END_CASE
END_METHOD

METHOD MS_SelectPath : BOOL
VAR_INPUT
END_VAR
IF M_SetNewPath() THEN
	eTXTDataExchangerState := TXT_DATA_EXCHANGER_METHOD_DONE;
	
END_IF
END_METHOD

METHOD PROTECTED MS_Uninitialized
;
END_METHOD

PROPERTY Name : STRING
GET
Name := sName;
END_GET
SET
sName := Name;
END_SET
END_PROPERTY

METHOD PROTECTED StateMachine
CASE eTXTDataExchangerState OF
	TXT_DATA_EXCHANGER_UNINITIALIZED:
		MS_Uninitialized();
		
	TXT_DATA_EXCHANGER_INITIALIZING:
		MS_Initializing();
		
	TXT_DATA_EXCHANGER_IDLE:
		MS_Idle();
		
	TXT_DATA_EXCHANGER_ADD_LOGS:
		MS_AddLogs();	
		
	TXT_DATA_EXCHANGER_SELECT_PATH:
		MS_SelectPath();			
		
	TXT_DATA_EXCHANGER_SEARCH_FOR_FILE:
		MS_SearchForFile();			
	
	TXT_DATA_EXCHANGER_RESET:
		MS_Reset();
		
	TXT_DATA_EXCHANGER_METHOD_DONE:
		MS_MethodDone();
	
	TXT_DATA_EXCHANGER_ABORTING:
		MS_Aborting();
	
END_CASE
END_METHOD

END_FUNCTION_BLOCK

// ---- POUs/Libs/Utilities/StringMerge/FUN_MergeStrings3.TcPOU
(* 
:Description: This function is used to merge 5 strings
*)
FUNCTION FUN_MergeStrings3 : STRING
VAR_INPUT
	sStr1	: STRING;			(* Fifth string in merge row *)
	sStr2	: STRING;			(* Fourth string in merge row *)
	sStr3	: STRING;			(* Fourth string in merge row *)

END_VAR

FUN_MergeStrings3 := CONCAT(sStr1,sStr2);
FUN_MergeStrings3 := CONCAT(FUN_MergeStrings3,sStr3);

END_FUNCTION

// ---- POUs/Libs/Utilities/StringMerge/FUN_MergeStrings10.TcPOU
(* 
:Description: This function is used to merge 10 strings
*)
FUNCTION FUN_MergeStrings10 : STRING
VAR_INPUT
	sStr1	: STRING;		(* First string in merge row *)
	sStr2	: STRING;		(* Second string in merge row *)
	sStr3	: STRING;		(* Third string in merge row *)
	sStr4	: STRING(500);	(* Fourth string in merge row *)
	sStr5	: STRING(500);	(* Fifth string in merge row *)
	sStr6	: STRING(500);	(* Sixth string in merge row *)
	sStr7	: STRING(500);	(* Seventh string in merge row *)
	sStr8	: STRING;		(* Eight string in merge row *)
	sStr9	: STRING;		(* Ninth string in merge row *)
	sStr10	: STRING;		(* Tenth string in merge row *)
	
END_VAR

FUN_MergeStrings10 := CONCAT(sStr1,sStr2);
FUN_MergeStrings10 := CONCAT(FUN_MergeStrings10,sStr3);
FUN_MergeStrings10 := CONCAT(FUN_MergeStrings10,sStr4);
FUN_MergeStrings10 := CONCAT(FUN_MergeStrings10,sStr5);
FUN_MergeStrings10 := CONCAT(FUN_MergeStrings10,sStr6);
FUN_MergeStrings10 := CONCAT(FUN_MergeStrings10,sStr7);
FUN_MergeStrings10 := CONCAT(FUN_MergeStrings10,sStr8);
FUN_MergeStrings10 := CONCAT(FUN_MergeStrings10,sStr9);
FUN_MergeStrings10 := CONCAT(FUN_MergeStrings10,sStr10);

END_FUNCTION

// ---- POUs/Libs/Platform/Universal Safety/FB_UniversalSafety.TcPOU
(* 
:Description: This function block is base for of machine safety module in all projects.
*)
FUNCTION_BLOCK ABSTRACT FB_UniversalSafety IMPLEMENTS I_UniversalSafety
VAR_INPUT
END_VAR
VAR_OUTPUT
END_VAR
VAR
	bInit		: BOOL;
	bAbort		: BOOL;
	bReset		: BOOL;
	
	bError 		: BOOL;
	iErrorID 	: UDINT;
END_VAR
(*
Version history:

+-------------+------------+----------------+----------+------------------------------------------+
|Date         | Version    | created under  | Author   | Remark                                   |
+=============+============+================+==========+==========================================+
|2022-02      | 1.0.0.0    | V3.1.4024.22   | ADBO     | Function block created                   |
+-------------+------------+----------------+----------+------------------------------------------+

*)

METHOD MR_Abort : BOOL
VAR_INPUT
END_VAR
END_METHOD

METHOD MR_FirstCycle : BOOL
VAR_INPUT
END_VAR
END_METHOD

METHOD MR_Init : BOOL
VAR_INPUT
END_VAR
END_METHOD

METHOD MR_Reset : BOOL
VAR_INPUT
END_VAR
END_METHOD

METHOD PROTECTED ABSTRACT MS_Initializing
VAR_INPUT
END_VAR
END_METHOD

METHOD PROTECTED ABSTRACT MS_ReadyInitialized
VAR_INPUT
END_VAR
END_METHOD

METHOD PROTECTED ABSTRACT MS_Reset
VAR_INPUT
END_VAR
END_METHOD

METHOD PROTECTED ABSTRACT MS_ResetDone
VAR_INPUT
END_VAR
END_METHOD

METHOD PROTECTED ABSTRACT MS_Running
VAR_INPUT
END_VAR
;
END_METHOD

METHOD PROTECTED ABSTRACT MS_Uninitialized
VAR_INPUT
END_VAR
END_METHOD

METHOD PROTECTED StateMachine
VAR_INPUT
END_VAR
END_METHOD

END_FUNCTION_BLOCK

// ---- POUs/Libs/Platform/Universal Visu/F_CloseDialog.TcPOU
FUNCTION F_CloseDialog : BOOL
VAR_INPUT
	sDialogName : STRING;
END_VAR
VAR
	pstClientData : POINTER TO VisuElems.VisuStructClientData;
	itfDialogManager : VisuElems.IDialogManager;
	itfMyDialog : VisuElems.IVisualisationDialog;
	stVisuRect : VisuElems.VisuStructSimpleRectangle;
END_VAR

VisuElems.VisuElemBase.g_ClientManager.BeginIteration();
pstClientData := VisuElems.VisuElemBase.g_ClientManager.GetNextClient();
WHILE pstClientData <> 0 DO
   IF pstClientData^.GlobalData.ClientType = VisuElems.Visu_ClientType.HMITargetVisualization THEN
      itfDialogManager := VisuElems.g_VisuManager.GetDialogManager();
      itfMyDialog := itfDialogManager.GetDialog(sDialogName);
      itfDialogManager.CloseDialog	(itfMyDialog, pstClientData);
   END_IF
   pstClientData := VisuElems.VisuElemBase.g_ClientManager.GetNextClient();
END_WHILE

END_FUNCTION

// ---- POUs/Libs/Platform/Universal Visu/F_OpenDialog.TcPOU
FUNCTION F_OpenDialog : BOOL
VAR_INPUT
	sDialogName : STRING;
END_VAR
VAR
	pstClientData : POINTER TO VisuElems.VisuStructClientData;
	itfDialogManager : VisuElems.IDialogManager;
	itfMyDialog : VisuElems.IVisualisationDialog;
	stVisuRect : VisuElems.VisuStructSimpleRectangle;
END_VAR

VisuElems.VisuElemBase.g_ClientManager.BeginIteration();
pstClientData := VisuElems.VisuElemBase.g_ClientManager.GetNextClient();
WHILE pstClientData <> 0 DO
   IF pstClientData^.GlobalData.ClientType = VisuElems.Visu_ClientType.HMITargetVisualization THEN
      itfDialogManager := VisuElems.g_VisuManager.GetDialogManager();
      itfMyDialog := itfDialogManager.GetDialog(sDialogName);
     // stVisuRect.ptTopLeft.iX := ANY_TO_INT(INT#0);
     // stVisuRect.ptTopLeft.iY := ANY_TO_INT(INT#0);
      //stVisuRect.ptBottomRight.iX := ANY_TO_INT(10);
     // stVisuRect.ptBottomRight.iY := ANY_TO_INT(10);
      itfDialogManager.OpenDialog(itfMyDialog, pstClientData, FALSE, ADR(stVisuRect));
   END_IF
   pstClientData := VisuElems.VisuElemBase.g_ClientManager.GetNextClient();
END_WHILE

END_FUNCTION

// ---- POUs/Libs/Utilities/Beckhoff UPS/CX2xxx/FB_UpsCx2xxx.TcPOU
(* 
:Description: This function block takes care of persistent data save for CX1914 UPS for CX2xxx PLC series
*)
FUNCTION_BLOCK FB_UpsCx2xxx EXTENDS FB_UniversalCxUps
VAR	
	(* Function blocks *)
	fbWritePersistentData	: WritePersistentData;	(*  *)
	fbGetUPSStatus			: FB_GetUPSStatus;		(*  *)
	
	(* Timers *)
	tonPowerOkTimerOn		: TON;					(*  *)
	
	(* Triggers *)
	rtPowerLostRTrigger		: R_TRIG;				(*  *)
END_VAR
(*

Version history:

+-------------+------------+----------------+----------+------------------------------------------+
|Date         | Version    | created under  | Author   | Remark                                   |
+=============+============+================+==========+==========================================+
|2021-11      | 1.0.0.0    | V3.1.4024.22   | ADBO     | Function block created                   |
+-------------+------------+----------------+----------+------------------------------------------+
|2022-01      | 1.1.0.0    | V3.1.4024.22   | ADBO     | Changed to extension of FB_UniversalCxUps|
+-------------+------------+----------------+----------+------------------------------------------+

*)

(* Read status *)
fbGetUPSStatus(bEnable := TRUE);

(* Check if power is ok *)
bPowerOk := (fbGetUPSStatus.stStatus.ePowerStatus = PowerOnLine);

(* Detect that power lost *)
rtPowerLostRTrigger(CLK := NOT bPowerOk);

(* Writte persistent only if power was ok for 10 sec and it is lost *)
fbWritePersistentData(	NETID	:= sNetID,
						PORT 	:= iPlcPort,
						TMOUT	:= tTimeout,
						START 	:= rtPowerLostRTrigger.Q AND tonPowerOkTimerOn.Q);
						
(* Timer of power OK to use in next loop *)
tonPowerOkTimerOn(IN := bPowerOk, PT := T#10S);

END_FUNCTION_BLOCK

// ---- POUs/Libs/Utilities/Beckhoff UPS/Universal CX/FB_UniversalCxUps.TcPOU
(* 
:Description:
*)
FUNCTION_BLOCK ABSTRACT FB_UniversalCxUps IMPLEMENTS I_UniversalCxUps
VAR
	bFirstCycle : BOOL := TRUE;
	
	(* Internal parameters *)
	sName 		: STRING;
	sNetID		: STRING;
	iPlcPort 	: UINT;
	tTimeout	: TIME;
	
	(* Internal status *)
	bPowerOk	: BOOL;
END_VAR
(*
Version history:

+-------------+------------+----------------+----------+------------------------------------------+
|Date         | Version    | created under  | Author   | Remark                                   |
+=============+============+================+==========+==========================================+
|2022-01      | 1.0.0.0    | V3.1.4024.22   | ADBO     | Function block created                   |
+-------------+------------+----------------+----------+------------------------------------------+

*)

METHOD MR_FirstCycle : BOOL
VAR_INPUT
	sName 		: STRING;
	sNetID		: STRING;
	iPlcPort 	: UINT;
	tTimeout	: TIME;
END_VAR
THIS^.sName := sName;
THIS^.sNetID := sNetID;
THIS^.iPlcPort := iPlcPort;
THIS^.tTimeout := tTimeout;
END_METHOD

PROPERTY Name : STRING
GET
Name := sName;
END_GET
SET
sName := Name;
END_SET
END_PROPERTY

PROPERTY NetId : STRING
GET
NetId := sNetID;
END_GET
SET
sNetId := NetId;
END_SET
END_PROPERTY

PROPERTY PlcPort : UINT
GET
PlcPort := iPlcPort;
END_GET
SET
iPlcPort := PlcPort;
END_SET
END_PROPERTY

PROPERTY PowerOk : REFERENCE TO BOOL
GET
PowerOk REF= bPowerOk;
END_GET
END_PROPERTY

PROPERTY Timeout : TIME
GET
Timeout := tTimeout;
END_GET
SET
tTimeout := Timeout;
END_SET
END_PROPERTY

END_FUNCTION_BLOCK

// ---- POUs/Libs/Utilities/Beckhoff UPS/CX5xxx/FB_UpsCx50xx.TcPOU
(* 
:Description: This function block takes care of persistent data save for 1 second UPS from CX50xx series 
*)
FUNCTION_BLOCK FB_UpsCx50xx  EXTENDS FB_UpsCx5xxx
VAR	
	fbSavePersistentData : FB_S_UPS; (*  *)
END_VAR
(*
Version history:

+-------------+------------+----------------+----------+------------------------------------------+
|Date         | Version    | created under  | Author   | Remark                                   |
+=============+============+================+==========+==========================================+
|2021-11      | 1.0.0.0    | V3.1.4024.22   | ADBO     | Function block created                   |
+-------------+------------+----------------+----------+------------------------------------------+
|2022-01      | 1.1.0.0    | V3.1.4024.22   | ADBO     | Changed to extension of FB_UpsCx5xxx     |
+-------------+------------+----------------+----------+------------------------------------------+

*)

IF bFirstCycle THEN
	bFirstCycle := FALSE;
	iUpsPort := 16#4A8;
END_IF

(* Save persistent data when an power failure occurred *)
fbSavePersistentData(	sNetID			:= sNetID,
						iPLCPort		:= iPlcPort,
						iUPSPort		:= iUpsPort,
						tTimeout		:= tTimeout,
						eUpsMode		:= eUpsMode,
						ePersistentMode	:= ePersistentMode,
						tRecoverTime 	:= tRecoverTime);

bPowerOk := NOT fbSavePersistentData.bPowerFailDetect;

END_FUNCTION_BLOCK

// ---- POUs/Libs/Utilities/Beckhoff UPS/CX5xxx/FB_UpsCx5xxx.TcPOU
(* 
:Description:
*)
FUNCTION_BLOCK ABSTRACT FB_UpsCx5xxx EXTENDS FB_UniversalCxUps IMPLEMENTS I_BeckhoffUpsCX5xxx
VAR
	(* Internal parameters*)
	iUpsPort				: UINT;													(*  *)
	tRecoverTime			: TIME 				:= T#15S;							(*  *)
	eUpsMode				: E_S_UPS_Mode		:= eSUPS_WrPersistData_NoShutdown;	(*  *)
	ePersistentMode			: E_PersistentMode	:= SPDM_2PASS; 						(*  *)
END_VAR
(*
Version history:

+-------------+------------+----------------+----------+------------------------------------------+
|Date         | Version    | created under  | Author   | Remark                                   |
+=============+============+================+==========+==========================================+
|2022-01      | 1.0.0.0    | V3.1.4024.22   | ADBO     | Function block created                   |
+-------------+------------+----------------+----------+------------------------------------------+

*)

PROPERTY PersistentMode : E_PersistentMode
GET
PersistentMode := ePersistentMode;
END_GET
SET
ePersistentMode := PersistentMode;
END_SET
END_PROPERTY

PROPERTY RecoverTime : Time
GET
RecoverTime := tRecoverTime;
END_GET
SET
tRecoverTime := RecoverTime;
END_SET
END_PROPERTY

PROPERTY UpsMode : E_S_UPS_Mode
GET
UpsMode := eUpsMode;
END_GET
SET
eUpsMode := UpsMode;
END_SET
END_PROPERTY

PROPERTY UpsPort : UINT
GET
UpsPort := iUpsPort;
END_GET
SET
iUpsPort := UpsPort;
END_SET
END_PROPERTY

END_FUNCTION_BLOCK

// ---- POUs/Libs/Utilities/Beckhoff UPS/CX5xxx/FB_UpsCx51xx.TcPOU
(* 
:Description: This function block takes care of persistent data save for 1 second UPS from CX51xx series 
*)
FUNCTION_BLOCK FB_UpsCx51xx EXTENDS FB_UpsCx5xxx
VAR
	fbSavePersistentData : FB_S_UPS_CX51x0;	(*  *)
END_VAR
(*
Version history:

+-------------+------------+----------------+----------+------------------------------------------+
|Date         | Version    | created under  | Author   | Remark                                   |
+=============+============+================+==========+==========================================+
|2021-11      | 1.0.0.0    | V3.1.4024.22   | ADBO     | Function block created                   |
+-------------+------------+----------------+----------+------------------------------------------+
|2022-01      | 1.1.0.0    | V3.1.4024.22   | ADBO     | Changed to extension of FB_UpsCx5xxx     |
+-------------+------------+----------------+----------+------------------------------------------+

*)

IF bFirstCycle THEN
	bFirstCycle := FALSE;
	iUpsPort := 16#588;
END_IF

(* Save persistent data when an power failure occurred *)
fbSavePersistentData(	sNetID			:= sNetID,
						iPLCPort		:= iPlcPort,
						iUPSPort		:= iUpsPort,
						tTimeout		:= tTimeout,
						eUpsMode		:= eUpsMode,
						ePersistentMode	:= ePersistentMode,
						tRecoverTime 	:= tRecoverTime);

bPowerOk := NOT fbSavePersistentData.bPowerFailDetect;

END_FUNCTION_BLOCK

// ---- POUs/Libs/Utilities/CSV Data Exchanger/FB_CSVDataExchanger.TcPOU
FUNCTION_BLOCK FB_CSVDataExchanger IMPLEMENTS I_CSVDataExchanger
VAR	
	(* First cycle parameters *)
	sAmsNetId								: T_AmsNetId := '';							(* TwinCAT system network address *)
	sFileDir								: T_MaxString;								(* CSV source file directory *)
	sFileName 								: T_MaxString;								(* CSV source file name *)
	sFilePath								: T_MaxString;								(* CSV source file whole path *)
	bChangeSeparatorToComma					: BOOL;										(* CSV field separator *)

	(* VALUES TEMPORARY HARDCODED - until the file creation function will be implemented *)
	bCreateFile								: BOOL := FALSE; 							
	bAddHeader								: BOOL := FALSE;
	                                    	
	(* Current time *)                  	
	stTime									: TIMESTRUCT;	(*  *)
	sTime									: STRING;		(*  *)
	sFileDate								: STRING;		
	
	(* Function block status flags and parameters *)
	bActive									: BOOL;
	bBusy									: BOOL;
	bError									: BOOL;
	iErrorId								: UDINT;
	                                    	
	(* Temporary data holders and auxiliary variables *)        	
	sCSVLine								: T_MaxString := ''; 						(* Single CSV text line (row, record), we are using string as record buffer (your are able to see read fields)  *)
	sCSVField								: T_MaxString := ''; 						(* Single CSV field value (column, record field) *)
	iRow	 								: UDINT 	:= 0;							(* Row number (record) *)
	iColumn									: UDINT 	:= 0;							(* Column number (record field) *)
	iMaxNumberOfColumns						: UDINT		:= 0;							(* Maximum number of open file columns *)
	hFile									: UINT		:= 0;							(* File handle of the source file *)
	
	(* MS_SelectRow variables *)
	sFieldToString							: T_MaxString := ''; 						(* Single CSV field value converted to string format *)          
	sValueToSearch							: T_MaxString := ''; 						(* Searched value *)
	iColumnToSearch 						: UDINT;
	ptArrParsedString						: POINTER TO ARRAY[0..iMAX_CSV_COLUMNS - 1] OF STRING(iMAX_CSV_FIELD_LENGTH);	(* Target PLC database *)
	sRowResult								: STRING;

	(* MS_SelectAll variables *)		
	ptArrDatabase							: POINTER TO ARRAY[0..iMAX_CSV_ROWS - 1, 0..iMAX_CSV_COLUMNS - 1] OF STRING(iMAX_CSV_FIELD_LENGTH);	(* Target PLC database *)
	
	(* State machines *) 	
	eCSVDataExchangerState					: E_CSVDataExchangerState;
	eCSVDataExchangerSelectRowState			: E_CSVDataExchangerSelectRowState;			(* Current state of camera initialization *)
	eCSVDataExchangerSelectAllState			: E_CSVDataExchangerSelectAllState;
	eCSVDataExchangerInsertIntoTableState	: E_CSVDataExchangerInsertIntoTableState;
	eCSVDataExchangerInitState				: E_CSVDataExchangerInitState;
	eCSVDataExchangerCountColumnsState		: E_CSVDataExchangerCountColumnsState;
	eCSVDataExchangerSetNewPathState		: E_CSVDataExchangerSetNewPathState;
	
	(* Function blocks - file handling *)
	fbFileOpen								: FB_FileOpen;								(* Opens file *)
	fbFileClose								: FB_FileClose;								(* Closes file *)
	fbFileGets								: FB_FileGets;								(* Reads one record (line) *)
	fbReader								: FB_CSVMemBufferReader;					(* Helper function block used to parse CSV data bytes (single record line) *)
	fbFilePuts								: FB_FilePuts;								(* Writes one record (line) *)
	fbWriter								: FB_CSVMemBufferWriter;					(* Helper function block used to create CSV data bytes (single record line) *)
  	fbCreateDir								: FB_CreateDir;
END_VAR

bActive := eCSVDataExchangerState >= CSV_DATA_EXCHANGER_READY;

IF fbMachineTime.bValid THEN
	stTime := fbMachineTime.systemTime;
	sTime := SYSTEMTIME_TO_STRING(stTime);
	
END_IF

StateMachine();

PROPERTY Active : REFERENCE TO BOOL
GET
Active REF= bActive;
END_GET
END_PROPERTY

PROPERTY Busy : REFERENCE TO BOOL
GET
Busy REF= bBusy;
END_GET
END_PROPERTY

PROPERTY Error : REFERENCE TO BOOL
GET
Error REF= bError;
END_GET
END_PROPERTY

PROPERTY ErrorID : REFERENCE TO UDINT
GET
ErrorID REF= iErrorID;
END_GET
END_PROPERTY

PROPERTY FileDir : STRING
GET
FileDir := sFileDir;
END_GET
SET
sFileDir := FileDir;
END_SET
END_PROPERTY

PROPERTY FileName : STRING
GET
FileName := sFileName;
END_GET
SET
sFileName := FileName;
END_SET
END_PROPERTY

METHOD M_CountMaxNumberOfColumns : BOOL
VAR_INPUT
END_VAR
CASE eCSVDataExchangerCountColumnsState OF
	CSV_DATA_EXCHANGER_COUNT_COLUMNS_OPEN_FILE:
		M_CountMaxNumberOfColumns := FALSE;
		
		hFile	:= 0;
		iRow	:= 0;
		iColumn	:= 0;
		sCSVField := '';
		sCSVLine := '';
		fbFileOpen(bExecute := FALSE);
		
		fbFileOpen(sNetId := sAmsNetId, 
					sPathName := sFilePath,
					nMode := FOPEN_MODEREAD OR FOPEN_MODETEXT,(* Open file in TEXT mode! *)
					ePath := PATH_GENERIC, bExecute := TRUE );
					
		eCSVDataExchangerCountColumnsState := CSV_DATA_EXCHANGER_COUNT_COLUMNS_WAIT_FOR_OPENING;

	CSV_DATA_EXCHANGER_COUNT_COLUMNS_WAIT_FOR_OPENING:
		fbFileOpen(bExecute := FALSE, 
					bError => bError, 
					nErrID => iErrorId, 
					hFile => hFile );
					
		IF NOT fbFileOpen.bBusy THEN
			IF NOT fbFileOpen.bError THEN
				eCSVDataExchangerCountColumnsState := CSV_DATA_EXCHANGER_COUNT_COLUMNS_READ_SINGLE_LINE;
				
			ELSE(* Error: file not found? *)
				eCSVDataExchangerCountColumnsState := CSV_DATA_EXCHANGER_COUNT_COLUMNS_READING_DONE;
				
			END_IF
		END_IF

	CSV_DATA_EXCHANGER_COUNT_COLUMNS_READ_SINGLE_LINE:
		fbFileGets(bExecute := FALSE);
		
		fbFileGets(sNetId := sAmsNetId, 
					hFile := hFile, 
					bExecute := TRUE);
					
		eCSVDataExchangerCountColumnsState := CSV_DATA_EXCHANGER_COUNT_COLUMNS_WAIT_FOR_READING;

	CSV_DATA_EXCHANGER_COUNT_COLUMNS_WAIT_FOR_READING:
		fbFileGets(bExecute := FALSE, 
					bError => bError, 
					nErrID => iErrorId, 
					sLine => sCSVLine );
		
		IF NOT fbFileGets.bBusy THEN
			IF NOT fbFileGets.bError THEN
				IF NOT fbFileGets.bEOF THEN
					(* FB_FileGets returns text line without the CR (carriage return) character.
					We have to restore the CR character (replace the $L character with $R$L characters) *)
					IF RIGHT( sCSVLine, 1 ) = '$L' THEN
						sCSVLine := REPLACE(sCSVLine, '$R$L', 2, LEN(sCSVLine));
						
					END_IF
					eCSVDataExchangerCountColumnsState := CSV_DATA_EXCHANGER_COUNT_COLUMNS_COUNT;
					
				END_IF
			ELSE(* Error *)
				eCSVDataExchangerCountColumnsState := CSV_DATA_EXCHANGER_COUNT_COLUMNS_READING_DONE;
				
			END_IF
		END_IF

	CSV_DATA_EXCHANGER_COUNT_COLUMNS_COUNT:
		fbReader.eCmd := eEnumCmd_First;(* Read first field value *)
		
		REPEAT
			fbReader(pBuffer := ADR(sCSVLine), 
						cbBuffer := SIZEOF(sCSVLine), 
						getValue => sCSVField);
						
			IF fbReader.bOk THEN
				fbReader.eCmd := eEnumCmd_Next;(* Read next field value *)
				
				iColumn := iColumn + 1;(* Increment number of read columns *)
				
				IF fbReader.bCRLF THEN(* CRLF == TRUE => End of reacord reached *)
					iMaxNumberOfColumns := iColumn;(* Reset number of columns *)
					
				END_IF
			ELSE(* Error: End of record reached or all fields read *)
				eCSVDataExchangerCountColumnsState := CSV_DATA_EXCHANGER_COUNT_COLUMNS_CLOSE_FILE;
				
			END_IF
		UNTIL NOT fbReader.bOk
		END_REPEAT

	CSV_DATA_EXCHANGER_COUNT_COLUMNS_CLOSE_FILE:
		fbFileClose(bExecute := FALSE);
		
		fbFileClose(sNetId := sAmsNetId, 
					hFile := hFile, 
					bExecute := TRUE );
					
		eCSVDataExchangerCountColumnsState := CSV_DATA_EXCHANGER_COUNT_COLUMNS_WAIT_FOR_CLOSING;

	CSV_DATA_EXCHANGER_COUNT_COLUMNS_WAIT_FOR_CLOSING:
		fbFileClose(bExecute := FALSE, 
					bError => bError, 
					nErrID => iErrorId);
		
		IF NOT fbFileClose.bBusy THEN
			hFile := 0;
			eCSVDataExchangerCountColumnsState := CSV_DATA_EXCHANGER_COUNT_COLUMNS_READING_DONE;
			
		END_IF

	CSV_DATA_EXCHANGER_COUNT_COLUMNS_READING_DONE:
		IF (hFile <> 0) THEN
			eCSVDataExchangerCountColumnsState := CSV_DATA_EXCHANGER_COUNT_COLUMNS_CLOSE_FILE;
			
		ELSE
			hFile	:= 0;
			iRow	:= 0;
			iColumn	:= 0;
			sCSVField := '';
			sCSVLine := '';
			M_CountMaxNumberOfColumns := TRUE;
			eCSVDataExchangerCountColumnsState := CSV_DATA_EXCHANGER_COUNT_COLUMNS_OPEN_FILE;
			
		END_IF

END_CASE
END_METHOD

METHOD M_FieldSeparator : BOOL
VAR_INPUT
END_VAR
IF bChangeSeparatorToComma THEN
	DEFAULT_CSV_FIELD_SEP := 16#2C;(* Comma ASCII code *)
	
ELSE
	DEFAULT_CSV_FIELD_SEP := 16#3B;(* Semicolon ASCII code *)
	
END_IF

M_FieldSeparator := TRUE;
END_METHOD

METHOD M_FileProperties : BOOL
VAR_INPUT
END_VAR
IF NOT bCreateFile THEN
	bAddHeader := FALSE;

END_IF

M_FileProperties := TRUE;
END_METHOD

METHOD M_ResetParameters : BOOL
VAR_INPUT
END_VAR
fbCreateDir(bExecute := FALSE);
fbFileOpen(bExecute := FALSE);
fbFilePuts(bExecute := FALSE);
fbFileClose(bExecute := FALSE);
fbFileGets(bExecute := FALSE);	

iRow := 0;
iColumn := 0;
hFile := 0;
sCSVField := '';
sCSVLine := '';
sFieldToString	:= '';
sValueToSearch := '';
iColumnToSearch := 0;
sRowResult := '';

stTime.wDay 			:= 0;
stTime.wDayOfWeek 		:= 0;
stTime.wHour 			:= 0;
stTime.wMilliseconds 	:= 0;
stTime.wMinute 			:= 0;
stTime.wMonth 			:= 0;
stTime.wSecond 			:= 0;
stTime.wYear 			:= 0;

bError 		:= FALSE;
iErrorID 	:= 0;

eCSVDataExchangerInitState					:= 0;
eCSVDataExchangerSelectAllState				:= 0;
eCSVDataExchangerInsertIntoTableState		:= 0;

M_ResetParameters := TRUE;
END_METHOD

METHOD M_SetNewPath : BOOL
VAR_INPUT
END_VAR
CASE eCSVDataExchangerSetNewPathState OF
	CSV_DATA_EXCHANGER_SET_NEW_PATH_CHANGE_PATH:
		M_SetNewPath := FALSE;
		sFilePath := CONCAT(STR1 := sFileDir, STR2 := sFileName);
		sFilePath := CONCAT(STR1 := sFilePath, STR2 := WSTRING_TO_STRING(".csv"));
		
		iMaxNumberOfColumns := 0;
		eCSVDataExchangerSetNewPathState := CSV_DATA_EXCHANGER_SET_NEW_PATH_COUNT_FILE_COLUMNS;
	
	CSV_DATA_EXCHANGER_SET_NEW_PATH_COUNT_FILE_COLUMNS:
		IF M_CountMaxNumberOfColumns() THEN
			M_SetNewPath := TRUE;
			eCSVDataExchangerSetNewPathState := CSV_DATA_EXCHANGER_SET_NEW_PATH_CHANGE_PATH;
			
		END_IF
		
END_CASE
END_METHOD

METHOD MR_Abort : BOOL
IF eCSVDataExchangerState >= CSV_DATA_EXCHANGER_READY THEN
	bBusy := TRUE;
	MR_Abort := FALSE;
	eCSVDataExchangerState := CSV_DATA_EXCHANGER_ABORTING;
	
ELSIF eCSVDataExchangerState = CSV_DATA_EXCHANGER_UNINITIALIZED THEN
	bBusy := FALSE;
	MR_Abort := TRUE;
	
END_IF
END_METHOD

METHOD MR_CreateTable : BOOL
VAR_INPUT
	sFileName 								: T_MaxString;					(*  *)
	bAddHeader								: BOOL;
END_VAR
sCreateFilePath := CONCAT(STR1 := sFileDir, STR2 := sFileName);
END_METHOD

METHOD MR_FirstCycle : BOOL
VAR_INPUT
	sAmsNetId					: T_AmsNetId;	(* TwinCAT system network address *)
	sFileDir					: T_MaxString;	(* CSV source file path *)
	sFileName 					: T_MaxString;	(* CSV source file name *)
//	bCreateFile					: BOOL;			(* If true FB will create file under given path *)
//	bAddHeader					: BOOL;			(* If true there will be a header at the beginning of the doc *)
	bChangeSeparatorToComma		: BOOL;			(* In USA/UK the CSV field separator is a comma. In Germany and some other 
												   European countries the CSV field separator is a semicolon. *)
END_VAR
THIS^.sAmsNetId := sAmsNetId;
THIS^.sFileDir := sFileDir;
THIS^.sFileName := sFileName;
THIS^.bChangeSeparatorToComma := bChangeSeparatorToComma;
//THIS^.bCreateFile := bCreateFile;
//THIS^.bAddHeader := bAddHeader;

M_FieldSeparator();
M_SetNewPath();
//M_FileProperties();
END_METHOD

METHOD MR_Init : BOOL
VAR_INPUT
END_VAR
IF eCSVDataExchangerState = CSV_DATA_EXCHANGER_UNINITIALIZED THEN
	bBusy := TRUE;
	MR_Init := FALSE;
	eCSVDataExchangerState := CSV_DATA_EXCHANGER_INITIALIZING;
	
ELSIF eCSVDataExchangerState >= CSV_DATA_EXCHANGER_READY THEN
	bBusy := FALSE;
	MR_Init := TRUE;
	
END_IF
END_METHOD

METHOD MR_InsertIntoTable : BOOL
VAR_INPUT
END_VAR
IF bWrite THEN
	bWrite 	:= FALSE;
	bBusy 	:= TRUE;
	bError	:= FALSE;
	nErrId	:= 0;
	hFile	:= 0;
	nRow	:= 0;
	nColumn	:= 0;
	step 	:= 1;
END_IF
END_METHOD

METHOD MR_ParseString : BOOL
VAR_INPUT
	iColumnToParse			: UDINT;
	sStringToParse 			: STRING;
	iArrParsedStringAdr 	: PVOID;
END_VAR
IF eCSVDataExchangerState = CSV_DATA_EXCHANGER_IDLE THEN
	bBusy := TRUE;
	MR_ParseString := FALSE;
	THIS^.iColumnToParse := iColumnToParse;
	THIS^.sStringToParse := sStringToParse;
	ptArrParsedString := iArrParsedStringAdr;
	eCSVDataExchangerState := CSV_DATA_EXCHANGER_PARSE_STRING;
	
ELSIF eCSVDataExchangerState = CSV_DATA_EXCHANGER_METHOD_DONE THEN
	bBusy := FALSE;
	MR_ParseString := TRUE;
	
END_IF
END_METHOD

METHOD MR_Reset : BOOL
IF eCSVDataExchangerState >= CSV_DATA_EXCHANGER_IDLE AND eCSVDataExchangerState <> CSV_DATA_EXCHANGER_METHOD_DONE THEN
	bBusy := TRUE;
	MR_Reset := FALSE;
	eCSVDataExchangerState := CSV_DATA_EXCHANGER_RESET;
	
ELSIF eCSVDataExchangerState = CSV_DATA_EXCHANGER_METHOD_DONE THEN
	bBusy := FALSE;
	MR_Reset := TRUE;
	
END_IF
END_METHOD

METHOD MR_SelectAll : BOOL
VAR_INPUT
	iArrDataBaseAdr 		: PVOID; 		(* A pointer to the string array where the 100 records (max.) from CSV file table are stored *)
END_VAR
IF eCSVDataExchangerState = CSV_DATA_EXCHANGER_IDLE THEN
	bBusy := TRUE;
	MR_SelectAll := FALSE;
	ptArrDatabase := iArrDataBaseAdr;
	eCSVDataExchangerState := CSV_DATA_EXCHANGER_SELECT_ALL;
	
ELSIF eCSVDataExchangerState = CSV_DATA_EXCHANGER_METHOD_DONE THEN
	bBusy := FALSE;
	MR_SelectAll := TRUE;
	
END_IF
END_METHOD

METHOD MR_SelectPath : BOOL
VAR_INPUT
	sFileDir								: T_MaxString; 			(* CSV source file directory name *)
	sFileName 								: T_MaxString; 			(* CSV source file name *)
END_VAR
IF eCSVDataExchangerState = CSV_DATA_EXCHANGER_IDLE THEN
	THIS^.sFileDir := sFileDir;	
	THIS^.sFileName := sFileName;	
	bBusy := TRUE;
	MR_SelectPath := FALSE;
	eCSVDataExchangerState := CSV_DATA_EXCHANGER_SELECT_PATH;
	
ELSIF eCSVDataExchangerState = CSV_DATA_EXCHANGER_METHOD_DONE THEN
	bBusy := FALSE;
	MR_SelectPath := TRUE;
	
END_IF
END_METHOD

METHOD MR_SelectRow : BOOL
VAR_INPUT
	iColumnToSearch 			: UDINT;		(* Column number to search the value in; columns are counted from 1 *)
	sValueToSearch				: STRING;		(* Value that you are looking for *)
	iArrParsedStringAdr 		: PVOID;		(* A pointer to the string array where the matched row with the search value is stored as a string array *)
END_VAR

VAR_OUTPUT
	sRowResult					: STRING;
END_VAR
IF eCSVDataExchangerState = CSV_DATA_EXCHANGER_IDLE THEN
	THIS^.sValueToSearch := sValueToSearch;
	IF iColumnToSearch > iMaxNumberOfColumns THEN
		iColumnToSearch := iMaxNumberOfColumns;
		
	END_IF
	THIS^.iColumnToSearch := iColumnToSearch - 1;
	THIS^.ptArrParsedString := iArrParsedStringAdr;
	bBusy := TRUE;
	MR_SelectRow := FALSE;
	eCSVDataExchangerState := CSV_DATA_EXCHANGER_SELECT_ROW;
	
ELSIF eCSVDataExchangerState = CSV_DATA_EXCHANGER_METHOD_DONE THEN
	sRowResult := THIS^.sRowResult;
	bBusy := FALSE;
	MR_SelectRow := TRUE;
	
END_IF
END_METHOD

METHOD PROTECTED MS_Aborting
IF M_ResetParameters() THEN
	eCSVDataExchangerState := CSV_DATA_EXCHANGER_UNINITIALIZED;
	
END_IF
END_METHOD

METHOD PROTECTED MS_Idle
VAR_INPUT
END_VAR
;
END_METHOD

METHOD PROTECTED MS_Initializing //C:\TwinCAT\log\filelog.txt
CASE eCSVDataExchangerInitState OF
	CSV_DATA_EXCHANGER_INIT_CREATE_DIR:
		IF bCreateFile THEN
			fbCreateDir(sNetId 		:= sAmsNetId,
						sPathName 	:= sFileDir,
						bExecute 	:= TRUE,
						tTimeout 	:= DEFAULT_ADS_TIMEOUT);
							
			IF NOT fbCreateDir.bBusy THEN
				eCSVDataExchangerInitState := CSV_DATA_EXCHANGER_INIT_GET_TIME;
				fbCreateDir(bExecute := FALSE);
				
			END_IF
		ELSE
			eCSVDataExchangerInitState := CSV_DATA_EXCHANGER_INIT_DONE;
			
		END_IF
		
	CSV_DATA_EXCHANGER_INIT_GET_TIME:
		IF fbMachineTime.bValid THEN
			stTime := fbMachineTime.systemTime;
			sTime := SYSTEMTIME_TO_STRING(stTime);
			sFileDate := LEFT(sTime,10);
			eCSVDataExchangerInitState := CSV_DATA_EXCHANGER_INIT_CREATE_FILE;
			
		END_IF
		
	CSV_DATA_EXCHANGER_INIT_CREATE_FILE:
		IF NOT fbFileOpen.bError THEN
			fbFileOpen(sNetId 		:= sAmsNetId,
						//sPathName 	:= FUN_MergeStrings5(sPathName,'','_',LEFT(sTime,10),'.csv'),
						sPathName 	:= sFilePath,
						bExecute 	:= TRUE,
						tTimeout	:= DEFAULT_ADS_TIMEOUT,
						nMode		:= FOPEN_MODEAPPEND OR FOPEN_MODEPLUS);
							
			IF NOT fbFileOpen.bBusy THEN
				hFile := fbFileOpen.hFile;
				fbFileOpen(bExecute := FALSE);		
				
				IF bAddHeader THEN 
					eCSVDataExchangerInitState := CSV_DATA_EXCHANGER_INIT_ADD_HEADER;
					
				ELSE
					eCSVDataExchangerInitState :=CSV_DATA_EXCHANGER_INIT_CLOSE_FILE;
					
				END_IF							
			END_IF
		ELSE
			bError := fbFileOpen.bError;
			iErrorID := fbFileOpen.nErrId;
			fbFileOpen(bExecute := FALSE);
			
		END_IF
		
	CSV_DATA_EXCHANGER_INIT_ADD_HEADER:
		IF NOT fbFilePuts.bError THEN
			fbFilePuts(	sNetId := sAmsNetId,
						hFile := hFile,
						sLine := CONCAT('----- Logger file initialized at ',CONCAT(LEFT(sTime,23),' ----- $n')),
						bExecute := TRUE,
						tTimeout := DEFAULT_ADS_TIMEOUT);

			IF NOT fbFilePuts.bBusy THEN
				eCSVDataExchangerInitState := CSV_DATA_EXCHANGER_INIT_CLOSE_FILE;
				fbFilePuts( bExecute := FALSE);
				
			END_IF	
		ELSE
			bError := fbFilePuts.bError;
			iErrorID := fbFilePuts.nErrId;
			fbFilePuts( bExecute := FALSE);
			
		END_IF
	
	CSV_DATA_EXCHANGER_INIT_CLOSE_FILE:
		IF NOT fbFileClose.bError THEN
			fbFileClose( sNetId 		:= sAmsNetId,
							hFile 		:= hFile,
							bExecute 	:= TRUE,
							tTimeout 	:= DEFAULT_ADS_TIMEOUT);
							
			IF NOT fbFileClose.bBusy THEN
				fbFileClose( bExecute := FALSE);
				eCSVDataExchangerInitState := CSV_DATA_EXCHANGER_INIT_DONE;

			END_IF
		ELSE
			fbFileClose(bExecute := FALSE);
			bError := fbFileClose.bError;
			iErrorID := fbFileClose.nErrId;
			
		END_IF
	
	CSV_DATA_EXCHANGER_INIT_DONE:
		IF M_CountMaxNumberOfColumns() THEN
			eCSVDataExchangerInitState := CSV_DATA_EXCHANGER_INIT_CREATE_DIR;
			eCSVDataExchangerState := CSV_DATA_EXCHANGER_READY;
			
		END_IF
		
END_CASE
END_METHOD

METHOD MS_MethodDone : BOOL
VAR_INPUT
END_VAR
IF NOT bBusy THEN
	eCSVDataExchangerState := CSV_DATA_EXCHANGER_IDLE;
	
END_IF
END_METHOD

METHOD PROTECTED MS_Ready
VAR_INPUT
END_VAR
eCSVDataExchangerState := CSV_DATA_EXCHANGER_IDLE;
END_METHOD

METHOD PROTECTED MS_Reset
VAR_INPUT
END_VAR
IF M_ResetParameters() THEN
	eCSVDataExchangerState := CSV_DATA_EXCHANGER_METHOD_DONE;
	
END_IF
END_METHOD

METHOD MS_SelectAll : BOOL
CASE eCSVDataExchangerSelectAllState OF
	CSV_DATA_EXCHANGER_SELECT_ALL_OPEN_FILE:
		hFile	:= 0;
		iRow	:= 0;
		iColumn	:= 0;
		fbFileOpen(bExecute := FALSE);
		
		fbFileOpen(sNetId := sAmsNetId, 
					sPathName := sFilePath,
					nMode := FOPEN_MODEREAD OR FOPEN_MODETEXT,(* Open file in TEXT mode! *)
					ePath := PATH_GENERIC, bExecute := TRUE );
					
		eCSVDataExchangerSelectAllState := CSV_DATA_EXCHANGER_SELECT_ALL_WAIT_FOR_OPENING;

	CSV_DATA_EXCHANGER_SELECT_ALL_WAIT_FOR_OPENING:
		fbFileOpen(bExecute := FALSE, 
					bError => bError, 
					nErrID => iErrorId, 
					hFile => hFile );
					
		IF NOT fbFileOpen.bBusy THEN
			IF NOT fbFileOpen.bError THEN
				eCSVDataExchangerSelectAllState := CSV_DATA_EXCHANGER_SELECT_ALL_READ_SINGLE_LINE;
				
			ELSE(* Error: file not found? *)
				eCSVDataExchangerSelectAllState := CSV_DATA_EXCHANGER_SELECT_ALL_READING_DONE;
				
			END_IF
		END_IF

	CSV_DATA_EXCHANGER_SELECT_ALL_READ_SINGLE_LINE:
		fbFileGets(bExecute := FALSE);
		
		fbFileGets(sNetId := sAmsNetId, 
					hFile := hFile, 
					bExecute := TRUE);
					
		eCSVDataExchangerSelectAllState := CSV_DATA_EXCHANGER_SELECT_ALL_WAIT_FOR_READING;

	CSV_DATA_EXCHANGER_SELECT_ALL_WAIT_FOR_READING:
		fbFileGets(bExecute := FALSE, 
					bError => bError, 
					nErrID => iErrorId, 
					sLine => sCSVLine );
		
		IF NOT fbFileGets.bBusy THEN
			IF NOT fbFileGets.bError THEN
				IF fbFileGets.bEOF THEN
					eCSVDataExchangerSelectAllState := CSV_DATA_EXCHANGER_SELECT_ALL_CLOSE_FILE; (* End of file reached => Close source file *)
				
				ELSE
					(* FB_FileGets returns text line without the CR (carriage return) character.
					We have to restore the CR character (replace the $L character with $R$L characters) *)
					IF RIGHT( sCSVLine, 1 ) = '$L' THEN
						sCSVLine := REPLACE(sCSVLine, '$R$L', 2, LEN(sCSVLine));
						
					END_IF
					eCSVDataExchangerSelectAllState := CSV_DATA_EXCHANGER_SELECT_ALL_PARSE_SINGLE_LINE;
					
				END_IF
			ELSE(* Error *)
				eCSVDataExchangerSelectAllState := CSV_DATA_EXCHANGER_SELECT_ALL_READING_DONE;
				
			END_IF
		END_IF

	CSV_DATA_EXCHANGER_SELECT_ALL_PARSE_SINGLE_LINE:
		fbReader.eCmd := eEnumCmd_First;(* Read first field value *)
		
		REPEAT
			fbReader(pBuffer := ADR(sCSVLine), 
						cbBuffer := SIZEOF(sCSVLine), 
						getValue => sCSVField);
						
			IF fbReader.bOk THEN
				fbReader.eCmd := eEnumCmd_Next;(* Read next field value *)

				IF iRow <= iMAX_CSV_ROWS AND iColumn <= iMAX_CSV_COLUMNS THEN
						ptArrDatabase^[iRow, iColumn] := CSVFIELD_TO_STRING(sCSVField, FALSE);(* TODO: Save or use the field value in your application *)
						
				END_IF
				
				iColumn := iColumn + 1;(* Increment number of read columns *)
				
				IF fbReader.bCRLF THEN(* CRLF == TRUE => End of reacord reached *)
					iRow := iRow + 1;(* Increment number of read records *)
					iColumn 	:= 0;(* Reset number of columns *)
					iRow := iRow MOD iMAX_CSV_ROWS;
					
				END_IF
			ELSE(* Error: End of record reached or all fields read *)
				eCSVDataExchangerSelectAllState := CSV_DATA_EXCHANGER_SELECT_ALL_READ_SINGLE_LINE;
				
			END_IF
		UNTIL NOT fbReader.bOk
		END_REPEAT

	CSV_DATA_EXCHANGER_SELECT_ALL_CLOSE_FILE:
		fbFileClose(bExecute := FALSE);
		
		fbFileClose(sNetId := sAmsNetId, 
					hFile := hFile, 
					bExecute := TRUE );
					
		eCSVDataExchangerSelectAllState := CSV_DATA_EXCHANGER_SELECT_ALL_WAIT_FOR_CLOSING;

	CSV_DATA_EXCHANGER_SELECT_ALL_WAIT_FOR_CLOSING:
		fbFileClose(bExecute := FALSE, 
					bError => bError, 
					nErrID => iErrorId);
		
		IF NOT fbFileClose.bBusy THEN
			hFile := 0;
			eCSVDataExchangerSelectAllState := CSV_DATA_EXCHANGER_SELECT_ALL_READING_DONE;
			
		END_IF

	CSV_DATA_EXCHANGER_SELECT_ALL_READING_DONE:
		IF (hFile <> 0) THEN
			eCSVDataExchangerSelectAllState := CSV_DATA_EXCHANGER_SELECT_ALL_CLOSE_FILE;
			
		ELSE
			eCSVDataExchangerSelectAllState := CSV_DATA_EXCHANGER_SELECT_ALL_OPEN_FILE;
			eCSVDataExchangerState := CSV_DATA_EXCHANGER_METHOD_DONE;
			
		END_IF

END_CASE
END_METHOD

METHOD MS_SelectPath : BOOL
VAR_INPUT
END_VAR
IF M_SetNewPath() THEN
	eCSVDataExchangerState := CSV_DATA_EXCHANGER_METHOD_DONE;
	
END_IF
END_METHOD

METHOD MS_SelectRow : BOOL
VAR
	iLoop 				: UDINT;
END_VAR
CASE eCSVDataExchangerSelectRowState OF
	CSV_DATA_EXCHANGER_SELECT_ROW_OPEN_FILE:
		sRowResult := ' ';
		hFile	:= 0;
		iRow	:= 0;
		iColumn	:= 0;
		fbFileOpen(bExecute := FALSE);
		
		fbFileOpen(sNetId := sAmsNetId, 
					sPathName := sFilePath,
					nMode := FOPEN_MODEREAD OR FOPEN_MODETEXT,(* Open file in TEXT mode! *)
					ePath := PATH_GENERIC, bExecute := TRUE );
					
		eCSVDataExchangerSelectRowState := CSV_DATA_EXCHANGER_SELECT_ROW_WAIT_FOR_OPENING;

	CSV_DATA_EXCHANGER_SELECT_ROW_WAIT_FOR_OPENING:
		fbFileOpen(bExecute := FALSE, 
					bError => bError, 
					nErrID => iErrorId, 
					hFile => hFile );
					
		IF NOT fbFileOpen.bBusy THEN
			IF NOT fbFileOpen.bError THEN
				eCSVDataExchangerSelectRowState := CSV_DATA_EXCHANGER_SELECT_ROW_READ_SINGLE_LINE;
				
			ELSE(* Error: file not found? *)
				eCSVDataExchangerSelectRowState := CSV_DATA_EXCHANGER_SELECT_ROW_READING_DONE;
				
			END_IF
		END_IF

	CSV_DATA_EXCHANGER_SELECT_ROW_READ_SINGLE_LINE:
		fbFileGets(bExecute := FALSE);
		
		fbFileGets(sNetId := sAmsNetId, 
					hFile := hFile, 
					bExecute := TRUE);
					
		eCSVDataExchangerSelectRowState := CSV_DATA_EXCHANGER_SELECT_ROW_WAIT_FOR_READING;

	CSV_DATA_EXCHANGER_SELECT_ROW_WAIT_FOR_READING:
		fbFileGets(bExecute := FALSE, 
					bError => bError, 
					nErrID => iErrorId, 
					sLine => sCSVLine );
		
		IF NOT fbFileGets.bBusy THEN
			IF NOT fbFileGets.bError THEN
				IF fbFileGets.bEOF THEN
					eCSVDataExchangerSelectRowState := CSV_DATA_EXCHANGER_SELECT_ROW_CLOSE_FILE; (* End of file reached => Close source file *)
				
				ELSE
					(* FB_FileGets returns text line without the CR (carriage return) character.
					We have to restore the CR character (replace the $L character with $R$L characters) *)
					IF RIGHT( sCSVLine, 1 ) = '$L' THEN
						sCSVLine := REPLACE(sCSVLine, '$R$L', 2, LEN(sCSVLine));
						
					END_IF
					eCSVDataExchangerSelectRowState := CSV_DATA_EXCHANGER_SELECT_ROW_PARSE_SINGLE_LINE;
					
				END_IF
			ELSE(* Error *)
				eCSVDataExchangerSelectRowState := CSV_DATA_EXCHANGER_SELECT_ROW_READING_DONE;
				
			END_IF
		END_IF

	CSV_DATA_EXCHANGER_SELECT_ROW_PARSE_SINGLE_LINE:
		fbReader.eCmd := eEnumCmd_First;(* Read first field value *)
		WHILE iColumn <= iColumnToSearch - 1 DO 
			fbReader(pBuffer := ADR(sCSVLine), 
			cbBuffer := SIZEOF(sCSVLine), 
			getValue => sCSVField);
			
			ptArrParsedString^[iColumn] := sCSVField;
			
			IF fbReader.bOk THEN
				iColumn := iColumn + 1;
				fbReader.eCmd := eEnumCmd_Next;(* Read next field value *)
			END_IF
			
		END_WHILE
		
		REPEAT
			fbReader(pBuffer := ADR( sCSVLine ), cbBuffer := SIZEOF( sCSVLine ), getValue => sCSVField);
			
			IF fbReader.bOk THEN
				fbReader.eCmd := eEnumCmd_Next;(* Read next field value *)
				
				sFieldToString := CSVFIELD_TO_STRING(sCSVField, FALSE);(* TODO: Save or use the field value in your application *)

				IF iRow <= iMAX_CSV_ROWS AND iColumn = iColumnToSearch AND sFieldToString = sValueToSearch THEN
					sRowResult := sCSVLine;
						
				END_IF
				
				ptArrParsedString^[iColumn] := sCSVField;
				iColumn := iColumn + 1;(* Increment number of read columns *)
				IF fbReader.bCRLF THEN(* CRLF == TRUE => End of reacord reached *)
					iRow := iRow + 1;(* Increment number of read records *)
					iColumn := 0;
					iRow := iRow MOD iMAX_CSV_ROWS;
					
				END_IF

			ELSE(* Error: End of record reached or all fields read *)
				IF (sRowResult = ' ') THEN
					eCSVDataExchangerSelectRowState := CSV_DATA_EXCHANGER_SELECT_ROW_READ_SINGLE_LINE;
					
				ELSE
					eCSVDataExchangerSelectRowState := CSV_DATA_EXCHANGER_SELECT_ROW_CLOSE_FILE;
					
				END_IF
			END_IF
		UNTIL NOT fbReader.bOk
		END_REPEAT

	CSV_DATA_EXCHANGER_SELECT_ROW_CLOSE_FILE:
		fbFileClose(bExecute := FALSE);
		
		fbFileClose(sNetId := sAmsNetId, 
					hFile := hFile, 
					bExecute := TRUE );
					
		eCSVDataExchangerSelectRowState := CSV_DATA_EXCHANGER_SELECT_ROW_WAIT_FOR_CLOSING;

	CSV_DATA_EXCHANGER_SELECT_ROW_WAIT_FOR_CLOSING:
		fbFileClose(bExecute := FALSE, 
					bError => bError, 
					nErrID => iErrorId);
		
		IF NOT fbFileClose.bBusy THEN
			hFile := 0;
			eCSVDataExchangerSelectRowState := CSV_DATA_EXCHANGER_SELECT_ROW_READING_DONE;
			
		END_IF

	CSV_DATA_EXCHANGER_SELECT_ROW_READING_DONE:
		IF (hFile <> 0) THEN
			eCSVDataExchangerSelectRowState := CSV_DATA_EXCHANGER_SELECT_ROW_CLOSE_FILE;
			
		ELSE
			eCSVDataExchangerSelectRowState := CSV_DATA_EXCHANGER_SELECT_ROW_OPEN_FILE;
			eCSVDataExchangerState := CSV_DATA_EXCHANGER_METHOD_DONE;
			
		END_IF

END_CASE
END_METHOD

METHOD PROTECTED MS_Uninitialized
;
END_METHOD

METHOD PROTECTED StateMachine
CASE eCSVDataExchangerState OF
	CSV_DATA_EXCHANGER_UNINITIALIZED:
		MS_Uninitialized();
		
	CSV_DATA_EXCHANGER_INITIALIZING:
		MS_Initializing();
		
	CSV_DATA_EXCHANGER_READY:
		MS_Ready();
		
	CSV_DATA_EXCHANGER_IDLE:
		MS_Idle();
		
	CSV_DATA_EXCHANGER_SELECT_ALL:
		MS_SelectAll();
	
//	CSV_DATA_EXCHANGER_INSERT_INTO_TABLE:
//		MS_InsertIntoTable();

	CSV_DATA_EXCHANGER_SELECT_ROW:
		MS_SelectRow();
	
	CSV_DATA_EXCHANGER_SELECT_PATH:
		MS_SelectPath();

//	CSV_DATA_EXCHANGER_PARSE_STRING:
//		MS_ParseString();
		
	CSV_DATA_EXCHANGER_RESET:
		MS_Reset();
		
	CSV_DATA_EXCHANGER_METHOD_DONE:
		MS_MethodDone();	

	CSV_DATA_EXCHANGER_ABORTING:
		MS_Aborting();		
END_CASE
END_METHOD

END_FUNCTION_BLOCK

// ---- POUs/Libs/Utilities/Math/FUN_Ceil.TcPOU
(* 
:Description: This function determines a integral value from a floating point number that is a fraction bigger than or equal that number
*)
FUNCTION FUN_Ceil : LREAL
VAR_INPUT
	lrValue : LREAL; (* Input value to round*)
END_VAR
VAR
	lrIntegral	: LREAL; (* Integral part of input value *)
	lrDecimal 	: LREAL; (* Decimal part of input value *)
END_VAR
(*
Version history:

+-------------+------------+----------------+----------+------------------------------------------+
|Date         | Version    | created under  | Author   | Remark                                   |
+=============+============+================+==========+==========================================+
|2022-04      | 1.0.0.0    | V3.1.4024.22   | ADBO     | Function created		                  |
+-------------+------------+----------------+----------+------------------------------------------+

*)

(* Get integral part *)
lrIntegral := TRUNC(lrValue);

(* Get decimal part *)
lrDecimal := FRAC(lrValue);

(*Check decimal value and set final result *)
IF lrDecimal <> 0.0 THEN
	FUN_Ceil := lrIntegral + 1.0;
ELSE
	FUN_Ceil := lrIntegral;
END_IF

END_FUNCTION

// ---- POUs/Libs/Utilities/Recipes Manager/FB_RecipeParameter.TcPOU
FUNCTION_BLOCK FB_RecipeParameter IMPLEMENTS I_RecipeParameter
VAR
	sName		: STRING;
	bValue 		: BOOL;
	iValue		: DINT;
	rValue		: REAL;
	sValue		: STRING;
	psFileValue	: POINTER TO STRING;
	eType		: E_VisuCtrlRecipeParameterType;
END_VAR

PROPERTY BitValue : REFERENCE TO BOOL
GET
BitValue REF= bValue;
END_GET
END_PROPERTY

PROPERTY DataType : REFERENCE TO E_VisuCtrlRecipeParameterType
GET
DataType REF= eType;
END_GET
END_PROPERTY

PROPERTY FileValue : REFERENCE TO STRING
GET
FileValue REF= psFileValue^;
END_GET
END_PROPERTY

PROPERTY IntValue : REFERENCE TO DINT
GET
IntValue REF= iValue;
END_GET
END_PROPERTY

METHOD MR_FirstCycle : BOOL
VAR_INPUT
	eType			: E_VisuCtrlRecipeParameterType;
	sName			: STRING;
	pFileValueAdr	: PVOID;
END_VAR
THIS^.eType := eType;
THIS^.sName := sName;
THIS^.psFileValue := pFileValueAdr;
END_METHOD

PROPERTY Name : REFERENCE TO STRING
GET
Name REF= sName;
END_GET
END_PROPERTY

PROPERTY RealValue : REFERENCE TO REAL
GET
RealValue REF= rValue;
END_GET
END_PROPERTY

PROPERTY StringValue : REFERENCE TO STRING
GET
StringValue REF= sValue;
END_GET
END_PROPERTY

END_FUNCTION_BLOCK

// ---- POUs/Libs/Utilities/StringMerge/FUN_MergeLongStrings10.TcPOU
(* 
:Description: This function is used to merge 10 long strings
*)
FUNCTION FUN_MergeLongStrings10 : STRING(2000)
VAR_INPUT
	sStr1	: STRING(2000);
	sStr2	: STRING(2000);
	sStr3	: STRING(2000);
	sStr4	: STRING(2000);
	sStr5	: STRING(2000);
	sStr6	: STRING(2000);
	sStr7	: STRING(2000);
	sStr8	: STRING(2000);
	sStr9	: STRING(2000);
	sStr10	: STRING(2000);
END_VAR
VAR
	sStrTemp1 :	STRING(2000);
	sStrTemp2 :	STRING(2000);
END_VAR
(*
Version history:

+-------------+------------+----------------+----------+------------------------------------------+
|Date         | Version    | created under  | Author   | Remark                                   |
+=============+============+================+==========+==========================================+
|2021-11      | 1.0.0.0    | V3.1.4024.22   | ADBO     | Function created		                  |
+-------------+------------+----------------+----------+------------------------------------------+

*)

CONCAT2(ADR(sStr1),ADR(sStr2),ADR(sStrTemp1),SIZEOF(sStrTemp1));
CONCAT2(ADR(sStrTemp1),ADR(sStr3),ADR(sStrTemp2),SIZEOF(sStrTemp2));
CONCAT2(ADR(sStrTemp2),ADR(sStr4),ADR(sStrTemp1),SIZEOF(sStrTemp1));
CONCAT2(ADR(sStrTemp1),ADR(sStr5),ADR(sStrTemp2),SIZEOF(sStrTemp2));
CONCAT2(ADR(sStrTemp2),ADR(sStr6),ADR(sStrTemp1),SIZEOF(sStrTemp1));
CONCAT2(ADR(sStrTemp1),ADR(sStr7),ADR(sStrTemp2),SIZEOF(sStrTemp2));
CONCAT2(ADR(sStrTemp2),ADR(sStr8),ADR(sStrTemp1),SIZEOF(sStrTemp1));
CONCAT2(ADR(sStrTemp1),ADR(sStr9),ADR(sStrTemp2),SIZEOF(sStrTemp2));
CONCAT2(ADR(sStrTemp2),ADR(sStr10),ADR(FUN_MergeLongStrings10),SIZEOF(FUN_MergeLongStrings10));

END_FUNCTION

// ---- POUs/Libs/Vision/Cognex/FB_CognexCamera.TcPOU
FUNCTION_BLOCK FB_CognexCamera IMPLEMENTS I_CognexCamera
VAR
	bFirstCycle 						: BOOL := TRUE;				(* First cycle bit *)		
	sName 								: STRING;					(* TCP/IP device name for other utilities *)	
 	                        			
	(* Internal status *)   			
	bActive								: BOOL;						(* TCP/IP device initialized and ready to work *)
	bBusy								: BOOL;						(* TCP/IP device is currently proccesing *)
	bError								: BOOL;						(* Error occured while executing *)
	iErrorID 							: UDINT;					(* Error ID*)
	                        			
	eCameraState		 				: E_CognexCameraState;			(* Current state of camera connection *)
	eCameraInitState					: E_CognexCameraInitState;		(* Current state of camera initialization *)
	eCameraMethodState					: E_CognexCameraMethodState;
	eCameraGetPositionState				: E_CognexCameraGetPositionState;
	eCameraGetValuesState				: E_CognexCameraGetValuesState;
	                        	
	bConnectionLostError 				: BOOL;						(* Internal data exchange error - occured only in Running state *)
	
	eCameraGetConnectionStatus			: E_CognexCameraGetConnectionStatus;
	eCameraGetExprStatus				: E_CognexCameraGetExprStatus;
	eCameraGetFileListStatus			: E_CognexCameraGetFileListStatus;
	eCameraGetFileStatus				: E_CognexCameraGetFileStatus;
	eCameraGetJobStatus 				: E_CognexCameraGetJobStatus;
	eCameraGetOnlineStatus				: E_CognexCameraGetOnlineStatus;
	eCameraGetValueEasyBuilderStatus	: E_CognexCameraGetValueEasyBuilderStatus;
	eCameraGetValueSpreadsheetStatus	: E_CognexCameraGetValueSpreadsheetStatus;
	eCameraGetValueStatus				: E_CognexCameraGetValueStatus;
	eCameraLoadFileStatus				: E_CognexCameraLoadFileStatus;
	eCameraPutLiveStatus				: E_CognexCameraPutLiveStatus;
	eCameraPutPortnumStatus				: E_CognexCameraPutPortnumStatus;
	eCameraPutTimeoutStatus				: E_CognexCameraPutTimeoutStatus;
	eCameraPutUpdateStatus				: E_CognexCameraPutUpdateStatus;
	eCameraPutWatchStatus				: E_CognexCameraPutWatchStatus;
	eCameraResetSystemStatus			: E_CognexCameraResetSystemStatus;
	eCameraSetJobStatus					: E_CognexCameraSetJobStatus;
	eCameraSetOnlineStatus				: E_CognexCameraSetOnlineStatus;
	eCameraStoreFileStatus				: E_CognexCameraStoreFileStatus;
	eCameraGetPositionStatus			: E_CognexCameraGetPositionStatus;
	eCameraImageTriggerStatus			: E_CognexCameraImageTriggerStatus;
	eCameraGetValuesStatus				: E_CognexCameraGetValuesStatus;
	
	(* Function blocks *)
	fbTcpClient 						: FB_TcpClient;				(* FB to create client connection*)
	
	(* Timers *)
	tTimeout							: TON;
	
	(* Messages buffers *)
	stSendData							: ST_TcpBufferData;		(*  *)
	stReciveData 						: ST_TcpBufferData;		(*  *)

	(* Temporary messeges *)
	sSendMessage 						: STRING;				(*  *)
	sReciveMessage						: STRING(1000);			(*  *)
	arrBufferMessage					: ARRAY[0..10] OF STRING;
	iMessageIndex	 					: INT;	
	sNewLine							: STRING := '$R$L';
	
	(* Rising edge trigger *)
	rtError								: R_TRIG; 					(* Rising edge trigger for function block error *)
	
	(* Status inormation and number *)
	iLastStatusCode						: INT; 
	sLastStatusCode						: STRING;
	                        			
	sPositionXVariable					: STRING;
	sPositionYVariable					: STRING;
	sRotationVariable					: STRING;
	                        			
	sVariable1							: STRING;
	sVariable2							: STRING;
	sVariable3							: STRING;
	sVariable4							: STRING;
	                        			
	lrPositionX							: LREAL;
	lrPositionY							: LREAL;
	lrRotation							: LREAL;
                            			
	lrValue1							: LREAL;
	lrValue2							: LREAL;
	lrValue3							: LREAL;
	lrValue4							: LREAL;
	                        			
	sPositionString						: STRING;
	sPositionStringDel					: STRING; 
	
	(* Internal variables of methods *)
	sCellIndexExpr						: STRING;
	iColumnExpr 						: INT;
	iRowExpr 							: INT;
	sEasyBuilderValueName				: STRING;
	iColumnValueSpreadsheet				: INT;
	iRowValueSpreadsheet				: INT;
	sLoadFileName						: STRING;
	bEnableLiveAcquisition				: INT;
	iPortNumber							: INT;
	iTimeout							: INT;	
	iUpdateNumber						: INT;
	iColumnPut 							: INT;
	iRowPut 							: INT;
	iOutputEnable						: INT;
	iJobNumber							: INT;
	bSetCameraOnline					: INT;
	sStoreFileName						: STRING;
END_VAR

(* First cycle procedure *)
IF bFirstCycle THEN
	bFirstCycle := FALSE;	
		
END_IF

bActive := eCameraState >= CAMERA_READY;

(* Report errors that occur *)
rtError(CLK:=bError);

IF rtError.Q THEN 
	fbMachineLogger.MR_AddLogs(FUN_MergeStrings5(sName, ' : Error occured (error ID: ', UDINT_TO_STRING(iErrorID), ')', ''));

END_IF

(* Execute TCP/IP FB and timers *)
tTimeout();
fbTcpClient();

(* Execute state machine *)
StateMachine();

PROPERTY Active : REFERENCE TO BOOL
GET
Active REF= bActive;
END_GET
END_PROPERTY

PROPERTY Busy : REFERENCE TO BOOL
GET
Busy REF= bBusy;
END_GET
END_PROPERTY

PROPERTY Error : REFERENCE TO BOOL
GET
Error REF= bError;
END_GET
END_PROPERTY

PROPERTY ErrorID : REFERENCE TO UDINT
GET
ErrorID REF= iErrorID;
END_GET
END_PROPERTY

METHOD M_ResetParameters : BOOL
VAR_INPUT
END_VAR
eCameraGetConnectionStatus			:= 2;
eCameraGetExprStatus				:= 2;
eCameraGetFileListStatus			:= 2;
eCameraGetFileStatus				:= 2;
eCameraGetJobStatus 				:= 2;
eCameraGetOnlineStatus				:= 2;
eCameraGetValueEasyBuilderStatus	:= 2;
eCameraGetValueSpreadsheetStatus	:= 2;
eCameraGetValueStatus				:= 2;
eCameraLoadFileStatus				:= 2;
eCameraPutLiveStatus				:= 2;
eCameraPutPortnumStatus				:= 2;
eCameraPutTimeoutStatus				:= 2;
eCameraPutUpdateStatus				:= 2;
eCameraPutWatchStatus				:= 2;
eCameraResetSystemStatus			:= 2;
eCameraSetJobStatus					:= 2;
eCameraSetOnlineStatus				:= 2;
eCameraStoreFileStatus				:= 2;
eCameraGetPositionStatus			:= 2;
eCameraImageTriggerStatus			:= 2;
eCameraGetValuesStatus				:= 2;

sSendMessage 						:= '';
sReciveMessage						:= '';
iMessageIndex	 					:= 0;	

(* Status inormation and number *)
iLastStatusCode						:= 0; 
sLastStatusCode						:= '';
	
(* Internal variables of methods *)
sCellIndexExpr						:= '';
iColumnExpr 						:= 0;
iRowExpr 							:= 0;
sEasyBuilderValueName				:= '';
iColumnValueSpreadsheet				:= 0;
iRowValueSpreadsheet				:= 0;
sLoadFileName						:= '';
bEnableLiveAcquisition				:= 0;
iPortNumber							:= 0;
iTimeout							:= 0;	
iUpdateNumber						:= 0;
iColumnPut 							:= 0;
iRowPut 							:= 0;
iOutputEnable						:= 0;
iJobNumber							:= 0;
bSetCameraOnline					:= 0;
sStoreFileName						:= '';
	
sPositionXVariable					:= '';
sPositionYVariable					:= '';
sRotationVariable					:= '';

sVariable1							:= '';
sVariable2							:= '';
sVariable3							:= '';
sVariable4							:= '';

lrPositionX							:= 0.0;
lrPositionY							:= 0.0;
lrRotation							:= 0.0;

lrValue1							:= 0.0;
lrValue2							:= 0.0;			
lrValue3							:= 0.0;
lrValue4							:= 0.0;

sPositionString						:= '';
sPositionStringDel					:= '';	

(* Internal status *)
bActive								:= 0;						(* TCP/IP device initialized and ready to work *)
bBusy								:= 0;						(* TCP/IP device is currently proccesing *)
bError								:= 0;						(* Error occured while executing *)
iErrorID 							:= 0;					(* Error ID*)

	
eCameraGetPositionState := 0;
eCameraGetValuesState := 0;
eCameraMethodState := 0;
eCameraInitState := 0;

M_ResetParameters := TRUE;
END_METHOD

METHOD MR_Abort : BOOL
VAR_INPUT
END_VAR
IF eCameraState >= CAMERA_READY THEN
	bBusy := TRUE;
	MR_Abort := FALSE;
	eCameraState := CAMERA_ABORTING;
	fbMachineLogger.MR_AddLogs(CONCAT(sName,' : abort requested'));	
	
ELSIF eCameraState = CAMERA_UNINITIALIZED THEN
	bBusy := FALSE;
	MR_Abort := TRUE;
	fbMachineLogger.MR_AddLogs(CONCAT(sName,' : abort done'));	
	
END_IF
END_METHOD

METHOD MR_FirstCycle : BOOL
VAR_INPUT
	sCameraName 	: STRING;		(*  *)
	sClientHost		: T_IPv4Addr;	(*  *)
	sClientAmsNetID : T_AmsNetID;	(*  *)
	iClientPort		: UINT;			(*  *)
	tTimeout		: TIME;			(*  *)
END_VAR
(* Set fixture name *)
THIS^.sName := sCameraName;

(* Set fixture server initial parameters *)
THIS^.fbTcpClient.MR_FirstCycle(	sName 		:= CONCAT('TCP/IP client of ',sCameraName),
									sHost		:= sClientHost,
									sAmsNetID	:= sClientAmsNetID,
									iPort 		:= iClientPort,
									tTimeout 	:= tTimeout);
END_METHOD

METHOD MR_GetConnections : BOOL
IF eCameraState = CAMERA_IDLE THEN
	bBusy := TRUE;
	MR_GetConnections := FALSE;
	eCameraState := CAMERA_GET_CONNECTIONS;
	fbMachineLogger.MR_AddLogs(CONCAT(sName,' : returning current connection information requested'));	
	
ELSIF eCameraState = CAMERA_METHOD_DONE THEN
	bBusy := FALSE;
	MR_GetConnections := TRUE;
	fbMachineLogger.MR_AddLogs(CONCAT(sName,' : returning current connection information done'));	
	
END_IF
END_METHOD

METHOD MR_GetExpr : BOOL
VAR_INPUT
	sCellIndexExpr	: STRING;
	iColumnExpr	: INT;
	iRowExpr	: INT;
END_VAR
IF eCameraState = CAMERA_IDLE THEN
	THIS^.sCellIndexExpr := sCellIndexExpr;
	THIS^.iColumnExpr	:= iColumnExpr;
	THIS^.iRowExpr	:= iRowExpr;	
	bBusy := TRUE;
	MR_GetExpr := FALSE;
	eCameraState := CAMERA_GET_EXPR;
	fbMachineLogger.MR_AddLogs(CONCAT(sName,' : returning the parameters or value stored in the cell requested'));	
	
ELSIF eCameraState = CAMERA_METHOD_DONE THEN
	bBusy := FALSE;
	MR_GetExpr := TRUE;
	fbMachineLogger.MR_AddLogs(CONCAT(sName,' : returning the parameters or value stored in the cell done'));	
	
END_IF
END_METHOD

METHOD MR_GetFile : BOOL
IF eCameraState = CAMERA_IDLE THEN
	bBusy := TRUE;
	MR_GetFile := FALSE;
	eCameraState := CAMERA_GET_FILE;
	fbMachineLogger.MR_AddLogs(CONCAT(sName,' : getting the filename of the active job requested'));	
	
ELSIF eCameraState = CAMERA_METHOD_DONE THEN
	bBusy := FALSE;
	MR_GetFile := TRUE;
	fbMachineLogger.MR_AddLogs(CONCAT(sName,' : getting the filename of the active job done'));	
	
END_IF
END_METHOD

METHOD MR_GetFileList : BOOL
IF eCameraState = CAMERA_IDLE THEN
	bBusy := TRUE;
	MR_GetFileList := FALSE;
	eCameraState := CAMERA_GET_FILE_LIST;
	fbMachineLogger.MR_AddLogs(CONCAT(sName,' : returning the number and names of files stored in memory requested'));	
	
ELSIF eCameraState = CAMERA_METHOD_DONE THEN
	bBusy := FALSE;
	MR_GetFileList := TRUE;
	fbMachineLogger.MR_AddLogs(CONCAT(sName,' : returning the number and names of files stored in memory done'));	
	
END_IF
END_METHOD

METHOD MR_GetJob : BOOL
IF eCameraState = CAMERA_IDLE THEN
	bBusy := TRUE;
	MR_GetJob := FALSE;
	eCameraState := CAMERA_GET_JOB;
	fbMachineLogger.MR_AddLogs(CONCAT(sName,' : returning a status code (ID) of the active job requested'));	
	
ELSIF eCameraState = CAMERA_METHOD_DONE THEN
	bBusy := FALSE;
	MR_GetJob := TRUE;
	fbMachineLogger.MR_AddLogs(CONCAT(sName,' : returning a status code (ID) of the active job done'));	
	
END_IF
END_METHOD

METHOD MR_GetOnline : BOOL
IF eCameraState = CAMERA_IDLE THEN
	bBusy := TRUE;
	MR_GetOnline := FALSE;
	eCameraState := CAMERA_GET_ONLINE;
	fbMachineLogger.MR_AddLogs(CONCAT(sName,' : returning the online state of the vision system requested'));	
	
ELSIF eCameraState = CAMERA_METHOD_DONE THEN
	bBusy := FALSE;
	MR_GetOnline := TRUE;
	fbMachineLogger.MR_AddLogs(CONCAT(sName,' :  returning the online state of the vision system done'));	
	
END_IF
END_METHOD

METHOD MR_GetPosition : BOOL
VAR_INPUT
	sPositionXVariable		: STRING;
	sPositionYVariable		: STRING;
	sRotationVariable		: STRING;
END_VAR

VAR_OUTPUT
	lrPositionX				: LREAL;
	lrPositionY				: LREAL;
	lrRotation				: LREAL;
END_VAR
IF eCameraState = CAMERA_IDLE THEN
	THIS^.sPositionXVariable := sPositionXVariable;
	THIS^.sPositionYVariable := sPositionYVariable;
	THIS^.sRotationVariable := sRotationVariable;
	bBusy := TRUE;
	MR_GetPosition := FALSE;
	eCameraState := CAMERA_GET_POSITION;
	fbMachineLogger.MR_AddLogs(CONCAT(sName,' : getting current position of the product requested'));	
	
ELSIF eCameraState = CAMERA_METHOD_DONE THEN
	lrPositionX := THIS^.lrPositionX;
	lrPositionY := THIS^.lrPositionY;
	lrRotation := THIS^.lrRotation;
	bBusy := FALSE;
	MR_GetPosition := TRUE;
	fbMachineLogger.MR_AddLogs(CONCAT(sName,' : getting current position of the product done'));	
	
END_IF
END_METHOD

METHOD MR_GetValueEasyBuilder : BOOL
VAR_INPUT
	sEasyBuilderValueName	: STRING;
END_VAR
IF eCameraState = CAMERA_IDLE THEN
	THIS^.sEasyBuilderValueName := sEasyBuilderValueName;
	bBusy := TRUE;
	MR_GetValueEasyBuilder := FALSE;
	eCameraState := CAMERA_GET_VALUE_EASY_BUILDER;
	fbMachineLogger.MR_AddLogs(CONCAT(sName,' : returning the tool result or job data in EasyBuilder requested'));	
	
ELSIF eCameraState = CAMERA_METHOD_DONE THEN
	bBusy := FALSE;
	MR_GetValueEasyBuilder := TRUE;
	fbMachineLogger.MR_AddLogs(CONCAT(sName,' : returning the tool result or job data in EasyBuilder done'));	
	
END_IF
END_METHOD

METHOD MR_GetValues : BOOL
VAR_INPUT
	sVariable1				: STRING;
	sVariable2				: STRING;
	sVariable3				: STRING;
	sVariable4				: STRING;
END_VAR

VAR_OUTPUT
	lrValue1				: LREAL;
	lrValue2				: LREAL;
	lrValue3				: LREAL;
	lrValue4				: LREAL;	
END_VAR
IF eCameraState = CAMERA_IDLE THEN
	THIS^.sVariable1 := sVariable1;
	THIS^.sVariable2 := sVariable2;
	THIS^.sVariable3 := sVariable3;
	THIS^.sVariable4 := sVariable4;
	bBusy := TRUE;
	MR_GetValues := FALSE;
	eCameraState := CAMERA_GET_VALUES;
	fbMachineLogger.MR_AddLogs(CONCAT(sName,' : getting values from camera requested'));	
	
ELSIF eCameraState = CAMERA_METHOD_DONE THEN
	lrValue1 := THIS^.lrValue1;
	lrValue2 := THIS^.lrValue2;
	lrValue3 := THIS^.lrValue3;
	lrValue4 := THIS^.lrValue4;
	bBusy := FALSE;
	MR_GetValues := TRUE;
	fbMachineLogger.MR_AddLogs(CONCAT(sName,' : getting values from camera done'));	
	
END_IF
END_METHOD

METHOD MR_GetValueSpreadsheet : BOOL
VAR_INPUT
	iColumnValueSpreadsheet		: INT;
	iRowValueSpreadsheet		: INT;
END_VAR
IF eCameraState = CAMERA_IDLE THEN
	THIS^.iColumnValueSpreadsheet := iColumnValueSpreadsheet;
	THIS^.iRowValueSpreadsheet := iRowValueSpreadsheet;
	bBusy := TRUE;
	MR_GetValueSpreadsheet := FALSE;
	eCameraState := CAMERA_GET_VALUE_SPREADSHEET;
	fbMachineLogger.MR_AddLogs(CONCAT(sName,' : returning the tool result or job data in the Spreadsheet requested'));	
	
ELSIF eCameraState = CAMERA_METHOD_DONE THEN
	bBusy := FALSE;
	MR_GetValueSpreadsheet := TRUE;
	fbMachineLogger.MR_AddLogs(CONCAT(sName,' : returning the tool result or job data in the Spreadsheet done'));	
	
END_IF
END_METHOD

METHOD MR_ImageTrigger : BOOL
IF eCameraState = CAMERA_IDLE THEN
	bBusy := TRUE;
	MR_ImageTrigger := FALSE;
	eCameraState := CAMERA_IMAGE_TRIGGER;
	fbMachineLogger.MR_AddLogs(CONCAT(sName,' : image trigger requested'));	
	
ELSIF eCameraState = CAMERA_METHOD_DONE THEN
	bBusy := FALSE;
	MR_ImageTrigger := TRUE;
	fbMachineLogger.MR_AddLogs(CONCAT(sName,' : image trigger done'));	
	
END_IF
END_METHOD

METHOD MR_Init : BOOL
IF eCameraState = CAMERA_UNINITIALIZED THEN
	bBusy := TRUE;
	MR_Init := FALSE;
	eCameraState := CAMERA_INITIALIZING;
	fbMachineLogger.MR_AddLogs(CONCAT(sName,' : initializing requested'));	
	
ELSIF eCameraState >= CAMERA_READY THEN
	bBusy := FALSE;
	MR_Init := TRUE;
	fbMachineLogger.MR_AddLogs(CONCAT(sName,' : initializing done'));	
	
END_IF
END_METHOD

METHOD MR_LoadFile : BOOL
VAR_INPUT
	sLoadFileName	: STRING;
END_VAR
IF eCameraState = CAMERA_IDLE THEN
	THIS^.sLoadFileName := sLoadFileName;
	bBusy := TRUE;
	MR_LoadFile := FALSE;
	eCameraState := CAMERA_LOAD_FILE;
	fbMachineLogger.MR_AddLogs(CONCAT(sName,' : loading the specified job from flash memory requested'));	

ELSIF eCameraState = CAMERA_METHOD_DONE THEN
	bBusy := FALSE;
	MR_LoadFile := TRUE;
	fbMachineLogger.MR_AddLogs(CONCAT(sName,' :  loading the specified job from flash memory done'));	
	
END_IF
END_METHOD

METHOD MR_PutLive : BOOL
VAR_INPUT
	bEnableLiveAcquisition : INT;
END_VAR
IF eCameraState = CAMERA_IDLE THEN
	THIS^.bEnableLiveAcquisition := bEnableLiveAcquisition;
	bBusy := TRUE;
	MR_PutLive := FALSE;
	eCameraState := CAMERA_PUT_LIVE;
	fbMachineLogger.MR_AddLogs(CONCAT(sName,' : turning live acquisition mode on or off requested'));	
	
ELSIF eCameraState = CAMERA_METHOD_DONE THEN
	bBusy := FALSE;
	MR_PutLive := TRUE;
	fbMachineLogger.MR_AddLogs(CONCAT(sName,' : turning live acquisition mode on or off done'));	
	
END_IF
END_METHOD

METHOD MR_PutPortnum : BOOL
VAR_INPUT
	iPortNumber : INT;
END_VAR
IF eCameraState = CAMERA_IDLE THEN
	THIS^.iPortNumber := iPortNumber;
	bBusy := TRUE;
	MR_PutPortnum := FALSE;
	eCameraState := CAMERA_PUT_PORTNUM;
	fbMachineLogger.MR_AddLogs(CONCAT(sName,' : specifying the communication port number requested'));	
	
ELSIF eCameraState = CAMERA_METHOD_DONE THEN
	bBusy := FALSE;
	MR_PutPortnum := TRUE;
	fbMachineLogger.MR_AddLogs(CONCAT(sName,' : specifying the communication port number done'));	
	
END_IF
END_METHOD

METHOD MR_PutTimeout : BOOL
VAR_INPUT
	iTimeout 	: INT;
END_VAR
IF eCameraState = CAMERA_IDLE THEN
	THIS^.iTimeout := iTimeout;
	bBusy := TRUE;
	MR_PutTimeout := FALSE;
	eCameraState := CAMERA_PUT_TIMEOUT;
	fbMachineLogger.MR_AddLogs(CONCAT(sName,' : specifying a port connection timeout requested'));	
	
ELSIF eCameraState = CAMERA_METHOD_DONE THEN
	bBusy := FALSE;
	MR_PutTimeout := TRUE;
	fbMachineLogger.MR_AddLogs(CONCAT(sName,' : specifying a port connection timeout done'));	
	
END_IF
END_METHOD

METHOD MR_PutUpdate : BOOL
VAR_INPUT
	iUpdateNumber 	: INT;
END_VAR
IF eCameraState = CAMERA_IDLE THEN
	THIS^.iUpdateNumber := iUpdateNumber;
	bBusy := TRUE;
	MR_PutUpdate := FALSE;
	eCameraState := CAMERA_PUT_UPDATE;
	fbMachineLogger.MR_AddLogs(CONCAT(sName,' : updating the GUI requested'));	
	
ELSIF eCameraState = CAMERA_METHOD_DONE THEN
	bBusy := FALSE;
	MR_PutUpdate := TRUE;
	fbMachineLogger.MR_AddLogs(CONCAT(sName,' : updating the GUI done'));	
	
END_IF
END_METHOD

METHOD MR_PutWatch : BOOL
VAR_INPUT
	iColumnPut 		: INT;
	iRowPut 		: INT;
	iOutputEnable	: INT;
END_VAR
IF eCameraState = CAMERA_IDLE THEN
	THIS^.iColumnPut := iColumnPut;
	THIS^.iRowPut := iRowPut;
	THIS^.iOutputEnable := iOutputEnable;
	bBusy := TRUE;
	MR_PutWatch := FALSE;
	eCameraState := CAMERA_PUT_WATCH;
	fbMachineLogger.MR_AddLogs(CONCAT(sName,' : returning the value contained in the specified cell each time the cell is updated requested'));	
	
ELSIF eCameraState = CAMERA_METHOD_DONE THEN
	bBusy := FALSE;
	MR_PutWatch := TRUE;
	fbMachineLogger.MR_AddLogs(CONCAT(sName,' : returning the value contained in the specified cell each time the cell is updated done'));	
	
END_IF
END_METHOD

METHOD MR_Reset : BOOL
IF eCameraState >= CAMERA_READY AND eCameraState <> CAMERA_METHOD_DONE THEN
	bBusy := TRUE;
	MR_Reset := FALSE;
	eCameraState := CAMERA_RESET;	
	fbMachineLogger.MR_AddLogs(CONCAT(sName,' : camera FB reset requested'));	
	
ELSIF eCameraState = CAMERA_METHOD_DONE THEN
	bBusy := FALSE;
	MR_Reset := TRUE;
	fbMachineLogger.MR_AddLogs(CONCAT(sName,' : camera FB reset done'));	
	
END_IF
END_METHOD

METHOD MR_ResetSystem : BOOL
IF eCameraState = CAMERA_IDLE THEN
	bBusy := TRUE;
	MR_ResetSystem := FALSE;
	eCameraState := CAMERA_RESET_SYSTEM;
	fbMachineLogger.MR_AddLogs(CONCAT(sName,' : resetting the In-Sight sensor requested'));	
	
ELSIF eCameraState = CAMERA_METHOD_DONE THEN
	bBusy := FALSE;
	MR_ResetSystem := TRUE;
	fbMachineLogger.MR_AddLogs(CONCAT(sName,' : resetting the In-Sight sensor done'));	
	
END_IF
END_METHOD

METHOD MR_SetJob : BOOL
VAR_INPUT
	iJobNumber 		: INT;
END_VAR
IF eCameraState = CAMERA_IDLE THEN
	THIS^.iJobNumber := iJobNumber;
	bBusy := TRUE;
	MR_SetJob := FALSE;
	eCameraState := CAMERA_SET_JOB;
	fbMachineLogger.MR_AddLogs(CONCAT(sName,' : loading a job from one of the job slots in flash memory on the In-Sight sensor requested'));	
	
ELSIF eCameraState = CAMERA_METHOD_DONE THEN
	bBusy := FALSE;
	MR_SetJob := TRUE;
	fbMachineLogger.MR_AddLogs(CONCAT(sName,' : loading a job from one of the job slots in flash memory on the In-Sight sensor done'));	
	
END_IF
END_METHOD

METHOD MR_SetOnline : BOOL
VAR_INPUT
	bSetCameraOnline	: INT;
END_VAR
IF eCameraState = CAMERA_IDLE THEN
	THIS^.bSetCameraOnline := bSetCameraOnline;
	bBusy := TRUE;
	MR_SetOnline := FALSE;
	eCameraState := CAMERA_SET_ONLINE;
	fbMachineLogger.MR_AddLogs(CONCAT(sName,' : setting the In-Sight sensor into Online or Offline mode requested'));	
	
ELSIF eCameraState = CAMERA_METHOD_DONE THEN
	bBusy := FALSE;
	MR_SetOnline := TRUE;
	fbMachineLogger.MR_AddLogs(CONCAT(sName,' : setting the In-Sight sensor into Online or Offline mode done'));	
	
END_IF
END_METHOD

METHOD MR_StoreFile : BOOL
VAR_INPUT
	sStoreFileName 	: STRING;
END_VAR
IF eCameraState = CAMERA_IDLE THEN
	THIS^.sStoreFileName := sStoreFileName;
	bBusy := TRUE;
	MR_StoreFile := FALSE;
	eCameraState := CAMERA_STORE_FILE;
	fbMachineLogger.MR_AddLogs(CONCAT(sName,' : saving the current job in flash memory on the In-Sight vision system requested'));	
	
ELSIF eCameraState = CAMERA_METHOD_DONE THEN
	bBusy := FALSE;
	MR_StoreFile := TRUE;
	fbMachineLogger.MR_AddLogs(CONCAT(sName,' : saving the current job in flash memory on the In-Sight vision system done'));	
	
END_IF
END_METHOD

METHOD PROTECTED MS_Aborting
fbTcpClient.MR_Abort();

IF NOT fbTcpClient.Active THEN 
	IF M_ResetParameters() THEN
		eCameraState := CAMERA_UNINITIALIZED;
		
	END_IF	
END_IF
END_METHOD

METHOD PROTECTED MS_GetConnections
CASE eCameraMethodState OF
	CAMERA_METHOD_SEND_COMMAND:
		MEMSET(ADR(sSendMessage),0,SIZEOF(sSendMessage));
		sSendMessage := 'Get Connections$R$L';
		FUN_StringToTcpBufferData(ADR(sSendMessage),ADR(stSendData));
		
		IF fbTcpClient.MR_AppendToSendBuffer(stSendData) THEN
			eCameraMethodState := CAMERA_METHOD_RECEIVE_RESPONSE;
							
		END_IF

	CAMERA_METHOD_RECEIVE_RESPONSE:
		stReciveData := fbTcpClient.NextRecivedMessage;
		
